# B&R Automation Studio project ACOPOStrak_DATech_Pilot (part 6)

#### Main.st
```iecst
PROGRAM _INIT
	currentProcess							:= E_PROCESS_Stage11;
	fbUserData.Axis							:= ADR(StStage[10].Shuttle);
	nextSlot 								:= ADR(StStage[11]);

	fbShuttleOutCheck.ProcessPoint			:= ADR(ptStage11);

	targetSlot ACCESS ADR(StStage[10]);
	shuttleID ACCESS ADR(interface.Trak.Data[0]);
END_PROGRAM

PROGRAM _CYCLIC
	IF gSim = TRUE THEN
		bBlockReadOnceAck := bBlockReadOnce;
		bBlockSendOnceAck := bBlockSendOnce;
		bBlockSendShuttleIDAck := bBlockSendShuttleID;

		IF interface.Trak.ShuttleArrived = TRUE THEN
			interface.Equipment.Ready 		:= FALSE;

			tmr.IN 							:= TRUE;
			tmr.PT 							:= T#1s;
		END_IF

		IF tmr.Q = TRUE THEN
			interface.Equipment.Done 		:= TRUE;
		END_IF

		IF interface.Trak.ShuttleArrived = FALSE THEN
			tmr.IN							:= FALSE;
			interface.Equipment.Ready 		:= TRUE;
			interface.Equipment.Done 		:= FALSE;
		END_IF

		tmr();
	END_IF

	IF targetSlot.Interface = E_SLOT_UNKNOWN THEN
		step 				:= 0;
	END_IF

	CASE step OF
		0:	(* Modbus Interface Initialize and Shuttle Check *)
			bBlockSendShuttleID					:= FALSE;
			bBlockSendOnce						:= FALSE;
			bBlockReadOnce						:= FALSE;

			//interface.Trak.ShuttleArrived		:= FALSE;

			IF targetSlot.Shuttle.controlif <> 0 AND bBlockSendOnceAck = FALSE AND bBlockReadOnceAck = FALSE AND bBlockSendShuttleIDAck = FALSE THEN
				step 							:= 10;
			END_IF

		10:	(* Read Shuttle Data from userData *)
			fbUserData.DataAddress 				:= ADR(userData);
			fbUserData.DataSize 				:= SIZEOF(userData);
			fbUserData.Mode						:= mcACPTRAK_USERDATA_GET;
			fbUserData.Execute 					:= TRUE;

			IF fbUserData.Done = TRUE THEN
				//End to Read Data fron user Data
				fbUserData.Execute 				:= FALSE;

				//Copy User Data to Modbus IO
				brsmemcpy(ADR(interface.Trak.Data[0]),ADR(userData.SerialNumber), 11);
				brsmemcpy(ADR(interface.Trak.Data2[0]),ADR(userData.Data[0]), SIZEOF(userData.Data));

				//Start to Write userdata to Modbus
				bBlockSendOnce					:= TRUE;
				bBlockSendShuttleID				:= TRUE;
				step 							:= 11;
			END_IF

		11: (* Check End of write to Modbus *)
			IF bBlockSendOnceAck AND bBlockSendShuttleIDAck THEN
				bBlockSendOnce					:= FALSE;
				bBlockSendShuttleID				:= FALSE;
				step							:= 20;
			END_IF

		20: (* Check Process Ready *)
			IF targetSlot.Interface = E_SLOT_PROCESS_READY THEN
				step 							:= 30;
			ELSIF targetSlot.Shuttle.controlif = 0 THEN
				step 							:= 0;
			END_IF

		30:	(* Check Assemble Status and Slot Status *)
			IF (gSts.AsmState = E_ASM_PROCESS OR gSts.AsmState = E_ASM_IDLE)
				AND targetSlot.Interface = E_SLOT_PROCESS_READY THEN
				interface.Trak.ShuttleArrived	:= TRUE;
				fbShuttleOutCheck.Enable		:= TRUE;
				step 							:= 100;
			END_IF

		100: (* Wait Proess End and Next Stage Ready *)
			IF interface.Equipment.Done = TRUE AND NextReady THEN
				//Start to Read Data from PLC
				bBlockReadOnce					:= TRUE;
				step 							:= 101;
			END_IF

		101:
			IF bBlockReadOnceAck = TRUE THEN
				// Save Current Process Status
				userData.ProcessStatus			:= currentProcess;

				// Read process data from PLC
				brsmemcpy(ADR(userData.Data[0]), ADR(interface.Equipment.Data2[0]), SIZEOF(interface.Equipment.Data2));

				// End to Read Data from PLC
				bBlockReadOnce					:= FALSE;
				step := 110;
			END_IF

		110: 	//Write User Data
			fbUserData.DataAddress 				:= ADR(userData);
			fbUserData.DataSize 				:= SIZE_OF_USERDATA;
			fbUserData.Mode						:= mcACPTRAK_USERDATA_SET;
			fbUserData.Execute 					:= TRUE;

			IF fbUserData.Done = TRUE THEN
				fbUserData.Execute 				:= FALSE;
				//	interface.Trak.ShuttleArrived 	:= FALSE;
				targetSlot.Interface 			:= E_SLOT_TAKEOUT_READY;
				targetSlot.NextStage			:= nextSlot;
				step 							:= 120;
			END_IF

		120: 	//Done Check
			IF interface.Equipment.Done = FALSE THEN
				step 						:= 0;
			END_IF
	END_CASE;

	IF fbShuttleOutCheck.EventCount > 0 THEN
		interface.Trak.ShuttleArrived	:= FALSE;
		fbShuttleOutCheck.Enable		:= FALSE;
	END_IF

	IF targetSlot.Shuttle.controlif = 0 AND shuttleID <> '' THEN
		brsmemset(ADR(interface.Trak.Data[0]),0,11);
	END_IF

	fbUserData();
	fbShuttleOutCheck();
	Timer();
	Timer2();

END_PROGRAM
```

### Program Logical/Source/Control/ifStage12 (IEC) - CCR 3

#### Main.st
```iecst
PROGRAM _INIT
	currentProcess							:= E_PROCESS_Stage12;
	fbUserData.Axis							:= ADR(StStage[11].Shuttle);
	nextSlot 								:= ADR(StStage[12]);

	fbShuttleOutCheck.ProcessPoint			:= ADR(ptStage12);

	targetSlot ACCESS ADR(StStage[11]);
	shuttleID ACCESS ADR(interface.Trak.Data[0]);
END_PROGRAM

PROGRAM _CYCLIC
	IF gSim = TRUE THEN
		bBlockReadOnceAck := bBlockReadOnce;
		bBlockSendOnceAck := bBlockSendOnce;
		bBlockSendShuttleIDAck := bBlockSendShuttleID;

		IF interface.Trak.ShuttleArrived = TRUE THEN
			interface.Equipment.Ready 		:= FALSE;

			tmr.IN 							:= TRUE;
			tmr.PT 							:= T#1s;
		END_IF

		IF tmr.Q = TRUE THEN
			interface.Equipment.Done 		:= TRUE;
		END_IF

		IF interface.Trak.ShuttleArrived = FALSE THEN
			tmr.IN							:= FALSE;
			interface.Equipment.Ready 		:= TRUE;
			interface.Equipment.Done 		:= FALSE;
		END_IF

		tmr();
	END_IF

	IF targetSlot.Interface = E_SLOT_UNKNOWN THEN
		step 				:= 0;
	END_IF

	CASE step OF
		0:	(* Modbus Interface Initialize and Shuttle Check *)
			bBlockSendShuttleID					:= FALSE;
			bBlockSendOnce						:= FALSE;
			bBlockReadOnce						:= FALSE;

			//interface.Trak.ShuttleArrived		:= FALSE;

			IF targetSlot.Shuttle.controlif <> 0 AND bBlockSendOnceAck = FALSE AND bBlockReadOnceAck = FALSE AND bBlockSendShuttleIDAck = FALSE THEN
				step 							:= 10;
			END_IF

		10:	(* Read Shuttle Data from userData *)
			fbUserData.DataAddress 				:= ADR(userData);
			fbUserData.DataSize 				:= SIZEOF(userData);
			fbUserData.Mode						:= mcACPTRAK_USERDATA_GET;
			fbUserData.Execute 					:= TRUE;

			IF fbUserData.Done = TRUE THEN
				//End to Read Data fron user Data
				fbUserData.Execute 				:= FALSE;

				//Copy User Data to Modbus IO
				brsmemcpy(ADR(interface.Trak.Data[0]),ADR(userData.SerialNumber), 11);
				brsmemcpy(ADR(interface.Trak.Data2[0]),ADR(userData.Data[0]), SIZEOF(userData.Data));

				//Start to Write userdata to Modbus
				bBlockSendOnce					:= TRUE;
				bBlockSendShuttleID				:= TRUE;
				step 							:= 11;
			END_IF

		11: (* Check End of write to Modbus *)
			IF bBlockSendOnceAck AND bBlockSendShuttleIDAck THEN
				bBlockSendOnce					:= FALSE;
				bBlockSendShuttleID				:= FALSE;
				step							:= 20;
			END_IF

		20: (* Check Process Ready *)
			IF targetSlot.Interface = E_SLOT_PROCESS_READY THEN
				step 							:= 30;
			ELSIF targetSlot.Shuttle.controlif = 0 THEN
				step 							:= 0;
			END_IF

		30:	(* Check Assemble Status and Slot Status *)
			IF (gSts.AsmState = E_ASM_PROCESS OR gSts.AsmState = E_ASM_IDLE)
				AND targetSlot.Interface = E_SLOT_PROCESS_READY THEN
				interface.Trak.ShuttleArrived	:= TRUE;
				fbShuttleOutCheck.Enable		:= TRUE;
				step 							:= 100;
			END_IF

		100: (* Wait Proess End and Next Stage Ready *)
			IF interface.Equipment.Done = TRUE AND NextReady THEN
				//Start to Read Data from PLC
				bBlockReadOnce					:= TRUE;
				step 							:= 101;
			END_IF

		101:
			IF bBlockReadOnceAck = TRUE THEN
				// Save Current Process Status
				userData.ProcessStatus			:= currentProcess;

				// Read process data from PLC
				brsmemcpy(ADR(userData.Data[0]), ADR(interface.Equipment.Data2[0]), SIZEOF(interface.Equipment.Data2));

				// End to Read Data from PLC
				bBlockReadOnce					:= FALSE;
				step := 110;
			END_IF

		110: 	//Write User Data
			fbUserData.DataAddress 				:= ADR(userData);
			fbUserData.DataSize 				:= SIZE_OF_USERDATA;
			fbUserData.Mode						:= mcACPTRAK_USERDATA_SET;
			fbUserData.Execute 					:= TRUE;

			IF fbUserData.Done = TRUE THEN
				fbUserData.Execute 				:= FALSE;
				//	interface.Trak.ShuttleArrived 	:= FALSE;
				targetSlot.Interface 			:= E_SLOT_TAKEOUT_READY;
				targetSlot.NextStage			:= nextSlot;
				step 							:= 120;
			END_IF

		120: 	//Done Check
			IF interface.Equipment.Done = FALSE THEN
				step 						:= 0;
			END_IF
	END_CASE;

	IF fbShuttleOutCheck.EventCount > 0 THEN
		interface.Trak.ShuttleArrived	:= FALSE;
		fbShuttleOutCheck.Enable		:= FALSE;
	END_IF

	IF targetSlot.Shuttle.controlif = 0 AND shuttleID <> '' THEN
		brsmemset(ADR(interface.Trak.Data[0]),0,11);
	END_IF

	fbUserData();
	fbShuttleOutCheck();
	Timer();
	Timer2();

END_PROGRAM
```

### Program Logical/Source/Control/if3D (IEC) - 3D scanner flying 

#### Main.st - Init, cyclic, exit code
```iecst
PROGRAM _INIT

	fbFlyStage.InPoint				:= ADR(pt3DIn);
	fbFlyStage.OutPoint				:= ADR(pt3DOut);
	fbFlyStage.MaximumShuttleCount	:= 1;
	fbFlyStage.InitShuttleCount		:= 1;

	fbTrig.ProcessPoint				:= ADR(pt3D);
	fbTrigInfo.ProcessPoint			:= ADR(pt3D);

	ShReadInfo.Axis	:= ADR(Axis);

	ShReadSectorPosInfo.Sector		:= ADR(SectorTrackAll);
	ShReadSectorPosInfo.Axis		:= ADR(Axis);

	fbUserData.Axis	:= ADR(fbTrigInfo.TrgPointInfo);

	shuttleID ACCESS ADR(interface.Trak.Data[0]);

	g3DStartPos	:= 10.52;
	g3DEndPos	:= 10.588;
	AddedTime	:= 14000; //140000

END_PROGRAM

PROGRAM _CYCLIC

	bModuleOK;
	bMovQuitFifoEmpty;
	bMovQuitFifoFull;
	bMovQuitTargetTimeVioloation;
	bMovQuitMaxFrequencyViolation;

	//////////////////////////////////////////////////////////////////////////////////
	// 3D scanner with DS1119 module
	//////////////////////////////////////////////////////////////////////////////////
//	MovTargetTime	:= MovTimeValid + AddedTime;

	IF gSts.AsmState = E_ASM_EMS OR gSts.AsmState = E_ASM_IDLE OR gSts.AsmState = E_ASM_INITIALIZATION THEN
		//	fbFlyStage.Enable	:= FALSE;
		Step				:= STEP_WAIT;
	ELSIF gSts.AsmState = E_ASM_PROCESS OR gSts.AsmState = E_ASM_MANUAL OR gSts.AsmState = E_ASM_ON THEN
		//	fbFlyStage.Enable	:= TRUE;
	END_IF

	CASE Step OF

		STEP_WAIT:
			IF fbTrigInfo.TrgPointInfo.Axis.controlif = 0 AND shuttleID <> '' THEN
				brsmemset(ADR(interface.Trak.Data[0]), 0, 11);
				userData.SerialNumber	:= '';
			END_IF

			interface.Trak.ShuttleArrived	:= FALSE;
			doTrigger						:= FALSE;
//			EncCnt							:= 0;
			IF gSts.AsmState = E_ASM_PROCESS OR gSts.AsmState = E_ASM_MANUAL OR gSts.AsmState = E_ASM_ON THEN
				fbTrig.Enable	:= TRUE;

				IF fbTrig.Valid THEN
					MovTargetPosition	:= LREAL_TO_DINT((g3DStartPos - 0.005) * 1000000);
					Step				:= STEP_IDLE;
				END_IF
			ELSE
				fbTrig.Enable	:= FALSE;
			END_IF

		STEP_IDLE:

			IF fbTrig.EventCount > 0 THEN
				fbTrigInfo.Execute	:= TRUE;

				fbUserData.DataAddress	:= ADR(userData);
				fbUserData.DataSize		:= SIZE_OF_USERDATA;
				fbUserData.Mode			:= mcACPTRAK_USERDATA_GET;
				fbUserData.Execute		:= TRUE;

				Step					:= STEP_GETSH;
			END_IF

		STEP_GETSH:
			IF fbTrigInfo.Done AND fbUserData.Done THEN
				interface.Trak.ShuttleArrived	:= TRUE;
				Axis							:= fbTrigInfo.TrgPointInfo.Axis;

				brsmemcpy(ADR(interface.Trak.Data[0]), ADR(userData.SerialNumber), 11);

				ShReadSectorPosInfo.Enable		:= TRUE;

				IF ShReadSectorPosInfo.Valid THEN
					Step			:= STEP_PRERUN;
					MovTargetTime	:= MovTimeValid + AddedTime;
				END_IF
			END_IF

		STEP_PRERUN:
			MovEnable			:= TRUE;
			MovTargetPosition	:= LREAL_TO_DINT((g3DStartPos - 0.005) * 1000000);
			MovTargetTime 		:= MovTargetTime + 2000;

			IF ShReadSectorPosInfo.Info.Position >= g3DStartPos - 0.005 THEN
				doTrigger	:= TRUE;
				Step		:= STEP_END;
			END_IF

//			IF EncCnt >= 1 THEN
//				IF ShReadSectorPosInfo.Info.Position < g3DStartPos - 0.005 THEN
//					MovTargetPosition	:= LREAL_TO_DINT((g3DStartPos - 0.005) * 1000000);
//				ELSE
//					MovTargetPosition	:= LREAL_TO_DINT((g3DStartPos - 0.005) * 1000000);
//				END_IF
//			END_IF
			//			EncCnt	:= EncCnt + 1;
//			MovEnable			:= TRUE;
//			MovTargetPosition	:= LREAL_TO_DINT(ShReadSectorPosInfo.Info.Position * 1000000);
			//			IF ShReadSectorPosInfo.Info.Position >= g3DStartPos THEN
//				doTrigger	:= TRUE;
//				Step		:= STEP_END;
//			END_IF

		STEP_END:
			MovTargetPosition	:= LREAL_TO_DINT(ShReadSectorPosInfo.Info.Position * 1000000);
			MovTargetTime 		:= MovTargetTime + 2000;

			IF ShReadSectorPosInfo.Info.Position >= g3DEndPos THEN
				ShReadSectorPosInfo.Enable		:= FALSE;
				interface.Trak.ShuttleArrived	:= FALSE;
				MovEnable						:= FALSE;
				doTrigger						:= FALSE;
				fbTrigInfo.Execute				:= FALSE;
				fbUserData.Execute				:= FALSE;
				Step							:= STEP_WAIT;
			END_IF

	END_CASE;

	// FB calls
	fbFlyStage();
	fbTrig();
	fbTrigInfo();
	fbUserData();
	ShReadSectorPosInfo();

END_PROGRAM
```

#### Variables.var - Local variables
```iecst
(**)
VAR
	MovEnable : BOOL;
	MovReset : BOOL;
	MovTargetPosition : DINT;
	MovTargetTime : DINT;
	MovPosition : DINT;
	MovTimeValid : DINT;
	AddedTime : DINT;
END_VAR
(**)
VAR
	nextReady : BOOL;
	shuttleID : REFERENCE TO STRING[19];
	userData : ShuttleUserData_typ;
	fbUserData : MC_BR_ShCopyUserData_AcpTrak;
END_VAR
(**)
VAR
	interface : Interface_Process_1Sh;
	fbFlyStage : MyTrak_TicketArea;
END_VAR
(**)
VAR
	fbTrigInfo : MC_BR_TrgPointGetInfo_AcpTrak;
	fbTrig : MC_BR_TrgPointEnable_AcpTrak;
	Axis : McAxisType;
	ShReadInfo : MC_BR_ShReadInfo_AcpTrak;
	ShReadSectorPosInfo : MC_BR_ShReadSectorPos_AcpTrak;
	Step : STEP_3DSensor;
	doTrigger : BOOL;
END_VAR
(**)
VAR
	timeMeasurement : TimingMeasurement_type;
END_VAR
(**)
VAR
	MoveTime : REAL;
	EncCnt : UINT;
END_VAR
(*Monitoring*)
VAR
	bModuleOK : BOOL;
	bMovQuitFifoEmpty : BOOL;
	bMovQuitFifoFull : BOOL;
	bMovQuitTargetTimeVioloation : BOOL;
	bMovQuitMaxFrequencyViolation : BOOL;
END_VAR
```

#### Types.typ
```iecst
TYPE
	STEP_3DSensor :
		(
		STEP_WAIT := 0,
		STEP_IDLE := 1,
		STEP_GETSH := 2,
		STEP_PRERUN := 3,
		STEP_END := 4
		);
	TimingMeasurement_type : 	STRUCT
		NextShuttle : MyTime_TimeCheck;
		ProcessingTime : MyTime_TimeCheck;
		MovementTime : MyTime_TimeCheck;
	END_STRUCT;
END_TYPE
```

### Program Logical/Source/Control/ifStage13 (IEC) - CCR 3

#### Main.st
```iecst
PROGRAM _INIT
	currentProcess							:= E_PROCESS_Stage13;
	fbUserData.Axis							:= ADR(StStage[12].Shuttle);
	nextSlot 								:= ADR(StStage[13]);

	fbShuttleOutCheck.ProcessPoint			:= ADR(ptStage13);

	targetSlot ACCESS ADR(StStage[12]);
	shuttleID ACCESS ADR(interface.Trak.Data[0]);

	NextReady 								:= TRUE;
END_PROGRAM

PROGRAM _CYCLIC
	IF gSim = TRUE THEN
		bBlockReadOnceAck := bBlockReadOnce;
		bBlockSendOnceAck := bBlockSendOnce;
		bBlockSendShuttleIDAck := bBlockSendShuttleID;

		IF interface.Trak.ShuttleArrived = TRUE THEN
			interface.Equipment.Ready 		:= FALSE;

			tmr.IN 							:= TRUE;
			tmr.PT 							:= T#1s;
		END_IF

		IF tmr.Q = TRUE THEN
			interface.Equipment.Done 		:= TRUE;
		END_IF

		IF interface.Trak.ShuttleArrived = FALSE THEN
			tmr.IN							:= FALSE;
			interface.Equipment.Ready 		:= TRUE;
			interface.Equipment.Done 		:= FALSE;
		END_IF

		tmr();
	END_IF

	IF targetSlot.Interface = E_SLOT_UNKNOWN THEN
		step 				:= 0;
	END_IF

	CASE step OF
		0:	(* Modbus Interface Initialize and Shuttle Check *)
			bBlockSendShuttleID					:= FALSE;
			bBlockSendOnce						:= FALSE;
			bBlockReadOnce						:= FALSE;

			//interface.Trak.ShuttleArrived		:= FALSE;

			IF targetSlot.Shuttle.controlif <> 0 AND bBlockSendOnceAck = FALSE AND bBlockReadOnceAck = FALSE AND bBlockSendShuttleIDAck = FALSE THEN
				step 							:= 10;
			END_IF

		10:	(* Read Shuttle Data from userData *)
			fbUserData.DataAddress 				:= ADR(userData);
			fbUserData.DataSize 				:= SIZEOF(userData);
			fbUserData.Mode						:= mcACPTRAK_USERDATA_GET;
			fbUserData.Execute 					:= TRUE;

			IF fbUserData.Done = TRUE THEN
				//End to Read Data fron user Data
				fbUserData.Execute 				:= FALSE;

				//Copy User Data to Modbus IO
				brsmemcpy(ADR(interface.Trak.Data[0]),ADR(userData.SerialNumber), 11);
				brsmemcpy(ADR(interface.Trak.Data2[0]),ADR(userData.Data[0]), SIZEOF(userData.Data));

				//Start to Write userdata to Modbus
				bBlockSendOnce					:= TRUE;
				bBlockSendShuttleID				:= TRUE;
				step 							:= 11;
			END_IF

		11: (* Check End of write to Modbus *)
			IF bBlockSendOnceAck AND bBlockSendShuttleIDAck THEN
				bBlockSendOnce					:= FALSE;
				bBlockSendShuttleID				:= FALSE;
				step							:= 20;
			END_IF

		20: (* Check Process Ready *)
			IF targetSlot.Interface = E_SLOT_PROCESS_READY THEN
				step 							:= 30;
			ELSIF targetSlot.Shuttle.controlif = 0 THEN
				step 							:= 0;
			END_IF

		30:	(* Check Assemble Status and Slot Status *)
			IF (gSts.AsmState = E_ASM_PROCESS OR gSts.AsmState = E_ASM_IDLE)
				AND targetSlot.Interface = E_SLOT_PROCESS_READY THEN
				interface.Trak.ShuttleArrived	:= TRUE;
				fbShuttleOutCheck.Enable		:= TRUE;
				step 							:= 100;
			END_IF

		100: (* Wait Proess End and Next Stage Ready *)
			IF interface.Equipment.Done = TRUE AND NextReady THEN
				//Start to Read Data from PLC
				bBlockReadOnce					:= TRUE;
				step 							:= 101;
			END_IF

		101:
			IF bBlockReadOnceAck = TRUE THEN
				// Save Current Process Status
				userData.ProcessStatus			:= currentProcess;

				// Read process data from PLC
				brsmemcpy(ADR(userData.Data[0]), ADR(interface.Equipment.Data2[0]), SIZEOF(interface.Equipment.Data2));

				// End to Read Data from PLC
				bBlockReadOnce					:= FALSE;
				step := 110;
			END_IF

		110: 	//Write User Data
			fbUserData.DataAddress 				:= ADR(userData);
			fbUserData.DataSize 				:= SIZE_OF_USERDATA;
			fbUserData.Mode						:= mcACPTRAK_USERDATA_SET;
			fbUserData.Execute 					:= TRUE;

			IF fbUserData.Done = TRUE THEN
				fbUserData.Execute 				:= FALSE;
				//	interface.Trak.ShuttleArrived 	:= FALSE;
				targetSlot.Interface 			:= E_SLOT_TAKEOUT_READY;
				targetSlot.NextStage			:= nextSlot;
				step 							:= 120;
			END_IF

		120: 	//Done Check
			IF interface.Equipment.Done = FALSE THEN
				step 						:= 0;
			END_IF
	END_CASE;

	IF fbShuttleOutCheck.EventCount > 0 THEN
		interface.Trak.ShuttleArrived	:= FALSE;
		fbShuttleOutCheck.Enable		:= FALSE;
	END_IF

	IF targetSlot.Shuttle.controlif = 0 AND shuttleID <> '' THEN
		brsmemset(ADR(interface.Trak.Data[0]),0,11);
	END_IF

	fbUserData();
	fbShuttleOutCheck();
	Timer();
	Timer2();

END_PROGRAM
```

### Program Logical/Source/Control/ifStage14 (IEC) - CSZ

#### Variables.var
```iecst
(**)
VAR
	currentProcess : E_PROCESS_STATUS;
	targetSlot : REFERENCE TO MyTrakSlotType;
	nextSlot : {REDUND_UNREPLICABLE} UDINT;
	shuttleID : REFERENCE TO STRING[19];
END_VAR
(**)
VAR
	step : DINT;
END_VAR
(**)
VAR
	interface : Interface_Process;
	userData : ShuttleUserData_typ;
END_VAR
(**)
VAR
	fbUserData : MC_BR_ShCopyUserData_AcpTrak;
END_VAR
(**)
VAR
	tmr : TON;
	fbShuttleOutCheck : MC_BR_TrgPointEnable_AcpTrak;
END_VAR
(**)
VAR
	NextReady : BOOL;
	Timer : TON;
	Timer2 : TON;
END_VAR
(**)
VAR
	bBlockSendOnce : BOOL;
	bBlockSendOnceAck : BOOL;
	bBlockReadOnce : BOOL;
	bBlockReadOnceAck : BOOL;
	bBlockSendShuttleID : BOOL;
	bBlockSendShuttleIDAck : BOOL;
END_VAR
(**)
VAR
	fbInterLock : MC_BR_BarrierCommand_AcpTrak;
	fbBarReadInfo : MC_BR_BarrierReadInfo_AcpTrak;
	ptInterlock : UDINT;
END_VAR
```

#### Main.st
```iecst
PROGRAM _INIT
	currentProcess							:= E_PROCESS_Stage14;
	fbUserData.Axis							:= ADR(StStage[13].Shuttle);
	nextSlot 								:= ADR(StStage[14]);

	fbShuttleOutCheck.ProcessPoint			:= ADR(ptStage14);

	ptInterlock								:= ADR(ptCSZInt);

	targetSlot ACCESS ADR(StStage[13]);
	shuttleID ACCESS ADR(interface.Trak.Data[0]);
END_PROGRAM

PROGRAM _CYCLIC
	IF gSim = TRUE THEN
		bBlockReadOnceAck := bBlockReadOnce;
		bBlockSendOnceAck := bBlockSendOnce;
		bBlockSendShuttleIDAck := bBlockSendShuttleID;

		IF interface.Trak.ShuttleArrived = TRUE THEN
			interface.Equipment.Ready 		:= FALSE;

			tmr.IN 							:= TRUE;
			tmr.PT 							:= T#1s;
		END_IF

		IF tmr.Q = TRUE THEN
			interface.Equipment.Done 		:= TRUE;
		END_IF

		IF interface.Trak.ShuttleArrived = FALSE THEN
			tmr.IN							:= FALSE;
			interface.Equipment.Ready 		:= TRUE;
			interface.Equipment.Done 		:= FALSE;
		END_IF

		tmr();
	END_IF

	//-----------------INTERLOCK--------------------
//	IF fbInterLock.Done = TRUE OR fbInterLock.Busy = TRUE OR fbInterLock.Error = TRUE THEN
//		fbInterLock.Execute 	:= FALSE;
//	ELSIF interface.Equipment.Ready = FALSE AND fbBarReadInfo.BarrierInfo.Status <> mcACPTRAK_BARRIER_CLOSED THEN
//		fbInterLock.Command 	:= mcACPTRAK_BARRIER_CLOSE;
//		fbInterLock.Execute 	:= TRUE;
//	ELSIF  interface.Equipment.Ready = TRUE AND fbBarReadInfo.BarrierInfo.Status <> mcACPTRAK_BARRIER_OPENED THEN
//		fbInterLock.Command 	:= mcACPTRAK_BARRIER_OPEN;
//		fbInterLock.Execute 	:= TRUE;
//	END_IF
//
//	fbBarReadInfo.Enable := TRUE;
//	fbBarReadInfo(ProcessPoint := ptInterlock);
//	fbInterLock(ProcessPoint := ptInterlock);
	//-----------------INTERLOCK--------------------

	IF targetSlot.Interface = E_SLOT_UNKNOWN THEN
		step 				:= 0;
	END_IF

	CASE step OF
		0:	(* Modbus Interface Initialize and Shuttle Check *)
			bBlockSendShuttleID					:= FALSE;
			bBlockSendOnce						:= FALSE;
			bBlockReadOnce						:= FALSE;

			//interface.Trak.ShuttleArrived		:= FALSE;

			IF targetSlot.Shuttle.controlif <> 0 AND bBlockSendOnceAck = FALSE AND bBlockReadOnceAck = FALSE AND bBlockSendShuttleIDAck = FALSE THEN
				step 							:= 10;
			END_IF

		10:	(* Read Shuttle Data from userData *)
			fbUserData.DataAddress 				:= ADR(userData);
			fbUserData.DataSize 				:= SIZEOF(userData);
			fbUserData.Mode						:= mcACPTRAK_USERDATA_GET;
			fbUserData.Execute 					:= TRUE;

			IF fbUserData.Done = TRUE THEN
				//End to Read Data fron user Data
				fbUserData.Execute 				:= FALSE;

				//Copy User Data to Modbus IO
				brsmemcpy(ADR(interface.Trak.Data[0]),ADR(userData.SerialNumber), 11);
				brsmemcpy(ADR(interface.Trak.Data2[0]),ADR(userData.Data[0]), SIZEOF(userData.Data));

				//Start to Write userdata to Modbus
				bBlockSendOnce					:= TRUE;
				bBlockSendShuttleID				:= TRUE;
				step 							:= 11;
			END_IF

		11: (* Check End of write to Modbus *)
			IF bBlockSendOnceAck AND bBlockSendShuttleIDAck THEN
				bBlockSendOnce					:= FALSE;
				bBlockSendShuttleID				:= FALSE;
				step							:= 20;
			END_IF

		20: (* Check Process Ready *)
			IF targetSlot.Interface = E_SLOT_PROCESS_READY THEN
				step 							:= 30;
			ELSIF targetSlot.Shuttle.controlif = 0 THEN
				step 							:= 0;
			END_IF

		30:	(* Check Assemble Status and Slot Status *)
			IF (gSts.AsmState = E_ASM_PROCESS OR gSts.AsmState = E_ASM_IDLE)
				AND targetSlot.Interface = E_SLOT_PROCESS_READY THEN
				interface.Trak.ShuttleArrived	:= TRUE;
				fbShuttleOutCheck.Enable		:= TRUE;
				step 							:= 100;
			END_IF

		100: (* Wait Proess End and Next Stage Ready *)
			IF interface.Equipment.Done = TRUE AND NextReady THEN
				//Start to Read Data from PLC
				bBlockReadOnce					:= TRUE;
				step 							:= 101;
			END_IF

		101:
			IF bBlockReadOnceAck = TRUE THEN
				// Save Current Process Status
				userData.ProcessStatus			:= currentProcess;

				// Read process data from PLC
				brsmemcpy(ADR(userData.Data[0]), ADR(interface.Equipment.Data2[0]), SIZEOF(interface.Equipment.Data2));

				// End to Read Data from PLC
				bBlockReadOnce					:= FALSE;
				step := 110;
			END_IF

		110: 	//Write User Data
			fbUserData.DataAddress 				:= ADR(userData);
			fbUserData.DataSize 				:= SIZE_OF_USERDATA;
			fbUserData.Mode						:= mcACPTRAK_USERDATA_SET;
			fbUserData.Execute 					:= TRUE;

			IF fbUserData.Done = TRUE THEN
				fbUserData.Execute 				:= FALSE;
				//	interface.Trak.ShuttleArrived 	:= FALSE;
				targetSlot.Interface 			:= E_SLOT_TAKEOUT_READY;
				targetSlot.NextStage			:= nextSlot;
				step 							:= 120;
			END_IF

		120: 	//Done Check
			IF interface.Equipment.Done = FALSE THEN
				step 						:= 0;
			END_IF
	END_CASE;

	IF fbShuttleOutCheck.EventCount > 0 THEN
		interface.Trak.ShuttleArrived	:= FALSE;
		fbShuttleOutCheck.Enable		:= FALSE;
	END_IF

	IF targetSlot.Shuttle.controlif = 0 AND shuttleID <> '' THEN
		brsmemset(ADR(interface.Trak.Data[0]),0,11);
	END_IF

	fbUserData();
	fbShuttleOutCheck();
	Timer();
	Timer2();

END_PROGRAM
```

### Program Logical/Source/Control/ifStage15 (IEC) - 3D arrive position

#### Main.st
```iecst
PROGRAM _INIT
	currentProcess							:= E_PROCESS_Stage15;
	fbUserData.Axis							:= ADR(StStage[14].Shuttle);
	nextSlot 								:= ADR(StStage[15]);

	fbShuttleOutCheck.ProcessPoint			:= ADR(ptStage15);

	targetSlot ACCESS ADR(StStage[14]);
	shuttleID ACCESS ADR(interface.Trak.Data[0]);
END_PROGRAM

PROGRAM _CYCLIC
	IF gSim = TRUE THEN
		bBlockReadOnceAck := bBlockReadOnce;
		bBlockSendOnceAck := bBlockSendOnce;
		bBlockSendShuttleIDAck := bBlockSendShuttleID;

		IF interface.Trak.ShuttleArrived = TRUE THEN
			interface.Equipment.Ready 		:= FALSE;

			tmr.IN 							:= TRUE;
			tmr.PT 							:= T#1s;
		END_IF

		IF tmr.Q = TRUE THEN
			interface.Equipment.Done 		:= TRUE;
		END_IF

		IF interface.Trak.ShuttleArrived = FALSE THEN
			tmr.IN							:= FALSE;
			interface.Equipment.Ready 		:= TRUE;
			interface.Equipment.Done 		:= FALSE;
		END_IF

		tmr();
	END_IF

	IF targetSlot.Interface = E_SLOT_UNKNOWN THEN
		step 				:= 0;
	END_IF

	CASE step OF
		0:	(* Modbus Interface Initialize and Shuttle Check *)
			bBlockSendShuttleID					:= FALSE;
			bBlockSendOnce						:= FALSE;
			bBlockReadOnce						:= FALSE;

			//interface.Trak.ShuttleArrived		:= FALSE;

			IF targetSlot.Shuttle.controlif <> 0 AND bBlockSendOnceAck = FALSE AND bBlockReadOnceAck = FALSE AND bBlockSendShuttleIDAck = FALSE THEN
				step 							:= 10;
			END_IF

		10:	(* Read Shuttle Data from userData *)
			fbUserData.DataAddress 				:= ADR(userData);
			fbUserData.DataSize 				:= SIZEOF(userData);
			fbUserData.Mode						:= mcACPTRAK_USERDATA_GET;
			fbUserData.Execute 					:= TRUE;

			IF fbUserData.Done = TRUE THEN
				//End to Read Data fron user Data
				fbUserData.Execute 				:= FALSE;

				//Copy User Data to Modbus IO
				brsmemcpy(ADR(interface.Trak.Data[0]),ADR(userData.SerialNumber), 11);
				brsmemcpy(ADR(interface.Trak.Data2[0]),ADR(userData.Data[0]), SIZEOF(userData.Data));

				//Start to Write userdata to Modbus
				bBlockSendOnce					:= TRUE;
				bBlockSendShuttleID				:= TRUE;
				step 							:= 11;
			END_IF

		11: (* Check End of write to Modbus *)
			IF bBlockSendOnceAck AND bBlockSendShuttleIDAck THEN
				bBlockSendOnce					:= FALSE;
				bBlockSendShuttleID				:= FALSE;
				step							:= 20;
			END_IF

		20: (* Check Process Ready *)
			IF targetSlot.Interface = E_SLOT_PROCESS_READY THEN
				step 							:= 30;
			ELSIF targetSlot.Shuttle.controlif = 0 THEN
				step 							:= 0;
			END_IF

		30:	(* Check Assemble Status and Slot Status *)
			IF (gSts.AsmState = E_ASM_PROCESS OR gSts.AsmState = E_ASM_IDLE)
				AND targetSlot.Interface = E_SLOT_PROCESS_READY THEN
				interface.Trak.ShuttleArrived	:= TRUE;
				fbShuttleOutCheck.Enable		:= TRUE;
				step 							:= 100;
			END_IF

		100: (* Wait Proess End and Next Stage Ready *)
			IF interface.Equipment.Done = TRUE AND NextReady THEN
				//Start to Read Data from PLC
				bBlockReadOnce					:= TRUE;
				step 							:= 101;
			END_IF

		101:
			IF bBlockReadOnceAck = TRUE THEN
				// Save Current Process Status
				userData.ProcessStatus			:= currentProcess;

				// Read process data from PLC
				brsmemcpy(ADR(userData.Data[0]), ADR(interface.Equipment.Data2[0]), SIZEOF(interface.Equipment.Data2));

				// End to Read Data from PLC
				bBlockReadOnce					:= FALSE;
				step := 110;
			END_IF

		110: 	//Write User Data
			fbUserData.DataAddress 				:= ADR(userData);
			fbUserData.DataSize 				:= SIZE_OF_USERDATA;
			fbUserData.Mode						:= mcACPTRAK_USERDATA_SET;
			fbUserData.Execute 					:= TRUE;

			IF fbUserData.Done = TRUE THEN
				fbUserData.Execute 				:= FALSE;
				//	interface.Trak.ShuttleArrived 	:= FALSE;
				targetSlot.Interface 			:= E_SLOT_TAKEOUT_READY;
				targetSlot.NextStage			:= nextSlot;
				step 							:= 120;
			END_IF

		120: 	//Done Check
			IF interface.Equipment.Done = FALSE THEN
				step 						:= 0;
			END_IF
	END_CASE;

	IF fbShuttleOutCheck.EventCount > 0 THEN
		interface.Trak.ShuttleArrived	:= FALSE;
		fbShuttleOutCheck.Enable		:= FALSE;
	END_IF

	IF targetSlot.Shuttle.controlif = 0 AND shuttleID <> '' THEN
		brsmemset(ADR(interface.Trak.Data[0]),0,11);
	END_IF

	fbUserData();
	fbShuttleOutCheck();
	Timer();
	Timer2();

END_PROGRAM
```

### Program Logical/Source/Control/ifStage16 (IEC) - Diameter inspection

#### Variables.var
```iecst
(**)
VAR
	currentProcess : E_PROCESS_STATUS;
	targetSlot : REFERENCE TO MyTrakSlotType;
	nextSlot : {REDUND_UNREPLICABLE} UDINT;
	shuttleID : REFERENCE TO STRING[19];
END_VAR
(**)
VAR
	step : DINT;
END_VAR
(**)
VAR
	interface : Interface_Process;
	userData : ShuttleUserData_typ;
END_VAR
(**)
VAR
	fbUserData : MC_BR_ShCopyUserData_AcpTrak;
END_VAR
(**)
VAR
	tmr : TON;
	fbShuttleOutCheck : MC_BR_TrgPointEnable_AcpTrak;
END_VAR
(**)
VAR
	NextReady : BOOL;
	Timer : TON;
	Timer2 : TON;
END_VAR
(**)
VAR
	bBlockSendOnce : BOOL;
	bBlockSendOnceAck : BOOL;
	bBlockReadOnce : BOOL;
	bBlockReadOnceAck : BOOL;
	bBlockSendShuttleID : BOOL;
	bBlockSendShuttleIDAck : BOOL;
END_VAR
```

#### Main.st
```iecst
PROGRAM _INIT
	currentProcess							:= E_PROCESS_Stage16;
	fbUserData.Axis							:= ADR(StStage[15].Shuttle);
	nextSlot 								:= ADR(StStage[16]);

	fbShuttleOutCheck.ProcessPoint			:= ADR(ptStage16);

	targetSlot ACCESS ADR(StStage[15]);
	shuttleID ACCESS ADR(interface.Trak.Data[0]);
END_PROGRAM

PROGRAM _CYCLIC
	IF gSim = TRUE THEN
		bBlockReadOnceAck := bBlockReadOnce;
		bBlockSendOnceAck := bBlockSendOnce;
		bBlockSendShuttleIDAck := bBlockSendShuttleID;

		IF interface.Trak.ShuttleArrived = TRUE THEN
			interface.Equipment.Ready 		:= FALSE;

			tmr.IN 							:= TRUE;
			tmr.PT 							:= T#1s;
		END_IF

		IF tmr.Q = TRUE THEN
			interface.Equipment.Done 		:= TRUE;
		END_IF

		IF interface.Trak.ShuttleArrived = FALSE THEN
			tmr.IN							:= FALSE;
			interface.Equipment.Ready 		:= TRUE;
			interface.Equipment.Done 		:= FALSE;
		END_IF

		tmr();
	END_IF

	IF targetSlot.Interface = E_SLOT_UNKNOWN THEN
		step 				:= 0;
	END_IF

	CASE step OF
		0:	(* Modbus Interface Initialize and Shuttle Check *)
			bBlockSendShuttleID					:= FALSE;
			bBlockSendOnce						:= FALSE;
			bBlockReadOnce						:= FALSE;

			//interface.Trak.ShuttleArrived		:= FALSE;

			IF targetSlot.Shuttle.controlif <> 0 AND bBlockSendOnceAck = FALSE AND bBlockReadOnceAck = FALSE AND bBlockSendShuttleIDAck = FALSE THEN
				step 							:= 10;
			END_IF

		10:	(* Read Shuttle Data from userData *)
			fbUserData.DataAddress 				:= ADR(userData);
			fbUserData.DataSize 				:= SIZEOF(userData);
			fbUserData.Mode						:= mcACPTRAK_USERDATA_GET;
			fbUserData.Execute 					:= TRUE;

			IF fbUserData.Done = TRUE THEN
				//End to Read Data fron user Data
				fbUserData.Execute 				:= FALSE;

				//Copy User Data to Modbus IO
				brsmemcpy(ADR(interface.Trak.Data[0]),ADR(userData.SerialNumber), 11);
				brsmemcpy(ADR(interface.Trak.Data2[0]),ADR(userData.Data[0]), SIZEOF(userData.Data));

				//Start to Write userdata to Modbus
				bBlockSendOnce					:= TRUE;
				bBlockSendShuttleID				:= TRUE;
				step 							:= 11;
			END_IF

		11: (* Check End of write to Modbus *)
			IF bBlockSendOnceAck AND bBlockSendShuttleIDAck THEN
				bBlockSendOnce					:= FALSE;
				bBlockSendShuttleID				:= FALSE;
				step							:= 20;
			END_IF

		20: (* Check Process Ready *)
			IF targetSlot.Interface = E_SLOT_PROCESS_READY THEN
				step 							:= 30;
			ELSIF targetSlot.Shuttle.controlif = 0 THEN
				step 							:= 0;
			END_IF

		30:	(* Check Assemble Status and Slot Status *)
			IF (gSts.AsmState = E_ASM_PROCESS OR gSts.AsmState = E_ASM_IDLE)
				AND targetSlot.Interface = E_SLOT_PROCESS_READY THEN
				interface.Trak.ShuttleArrived	:= TRUE;
				fbShuttleOutCheck.Enable		:= TRUE;
				step 							:= 100;
			END_IF

		100: (* Wait Proess End and Next Stage Ready *)
			IF interface.Equipment.Done = TRUE AND NextReady THEN
				//Start to Read Data from PLC
				bBlockReadOnce					:= TRUE;
				step 							:= 101;
			END_IF

		101:
			IF bBlockReadOnceAck = TRUE THEN
				// Save Current Process Status
				userData.ProcessStatus			:= currentProcess;

				// Read process data from PLC
				brsmemcpy(ADR(userData.Data[0]), ADR(interface.Equipment.Data2[0]), SIZEOF(interface.Equipment.Data2));

				// End to Read Data from PLC
				bBlockReadOnce					:= FALSE;
				step := 110;
			END_IF

		110: 	//Write User Data
			fbUserData.DataAddress 				:= ADR(userData);
			fbUserData.DataSize 				:= SIZE_OF_USERDATA;
			fbUserData.Mode						:= mcACPTRAK_USERDATA_SET;
			fbUserData.Execute 					:= TRUE;

			IF fbUserData.Done = TRUE THEN
				fbUserData.Execute 				:= FALSE;
				//	interface.Trak.ShuttleArrived 	:= FALSE;
				targetSlot.Interface 			:= E_SLOT_TAKEOUT_READY;
				targetSlot.NextStage			:= nextSlot;
				step 							:= 120;
			END_IF

		120: 	//Done Check
			IF interface.Equipment.Done = FALSE THEN
				step 						:= 0;
			END_IF
	END_CASE;

	IF fbShuttleOutCheck.EventCount > 0 THEN
		interface.Trak.ShuttleArrived	:= FALSE;
		fbShuttleOutCheck.Enable		:= FALSE;
	END_IF

	IF targetSlot.Shuttle.controlif = 0 AND shuttleID <> '' THEN
		brsmemset(ADR(interface.Trak.Data[0]),0,11);
	END_IF

	fbUserData();
	fbShuttleOutCheck();
	Timer();
	Timer2();

END_PROGRAM
```

### Program Logical/Source/Control/ifStage17 (IEC) - NG out

#### Main.st
```iecst
PROGRAM _INIT
	currentProcess							:= E_PROCESS_Stage17;
	fbUserData.Axis							:= ADR(StStage[16].Shuttle);
	nextSlot 								:= ADR(StStage[17]);

	fbShuttleOutCheck.ProcessPoint			:= ADR(ptStage17);

	targetSlot ACCESS ADR(StStage[16]);
	shuttleID ACCESS ADR(interface.Trak.Data[0]);
END_PROGRAM

PROGRAM _CYCLIC
	IF gSim = TRUE THEN
		bBlockReadOnceAck := bBlockReadOnce;
		bBlockSendOnceAck := bBlockSendOnce;
		bBlockSendShuttleIDAck := bBlockSendShuttleID;

		IF interface.Trak.ShuttleArrived = TRUE THEN
			interface.Equipment.Ready 		:= FALSE;

			tmr.IN 							:= TRUE;
			tmr.PT 							:= T#1s;
		END_IF

		IF tmr.Q = TRUE THEN
			interface.Equipment.Done 		:= TRUE;
		END_IF

		IF interface.Trak.ShuttleArrived = FALSE THEN
			tmr.IN							:= FALSE;
			interface.Equipment.Ready 		:= TRUE;
			interface.Equipment.Done 		:= FALSE;
		END_IF

		tmr();
	END_IF

	IF targetSlot.Interface = E_SLOT_UNKNOWN THEN
		step 				:= 0;
	END_IF

	CASE step OF
		0:	(* Modbus Interface Initialize and Shuttle Check *)
			bBlockSendShuttleID					:= FALSE;
			bBlockSendOnce						:= FALSE;
			bBlockReadOnce						:= FALSE;

			//interface.Trak.ShuttleArrived		:= FALSE;

			IF targetSlot.Shuttle.controlif <> 0 AND bBlockSendOnceAck = FALSE AND bBlockReadOnceAck = FALSE AND bBlockSendShuttleIDAck = FALSE THEN
				step 							:= 10;
			END_IF

		10:	(* Read Shuttle Data from userData *)
			fbUserData.DataAddress 				:= ADR(userData);
			fbUserData.DataSize 				:= SIZEOF(userData);
			fbUserData.Mode						:= mcACPTRAK_USERDATA_GET;
			fbUserData.Execute 					:= TRUE;

			IF fbUserData.Done = TRUE THEN
				//End to Read Data fron user Data
				fbUserData.Execute 				:= FALSE;

				//Copy User Data to Modbus IO
				brsmemcpy(ADR(interface.Trak.Data[0]),ADR(userData.SerialNumber), 11);
				brsmemcpy(ADR(interface.Trak.Data2[0]),ADR(userData.Data[0]), SIZEOF(userData.Data));

				//Start to Write userdata to Modbus
				bBlockSendOnce					:= TRUE;
				bBlockSendShuttleID				:= TRUE;
				step 							:= 11;
			END_IF

		11: (* Check End of write to Modbus *)
			IF bBlockSendOnceAck AND bBlockSendShuttleIDAck THEN
				bBlockSendOnce					:= FALSE;
				bBlockSendShuttleID				:= FALSE;
				step							:= 20;
			END_IF

		20: (* Check Process Ready *)
			IF targetSlot.Interface = E_SLOT_PROCESS_READY THEN
				step 							:= 30;
			ELSIF targetSlot.Shuttle.controlif = 0 THEN
				step 							:= 0;
			END_IF

		30:	(* Check Assemble Status and Slot Status *)
			IF (gSts.AsmState = E_ASM_PROCESS OR gSts.AsmState = E_ASM_IDLE)
				AND targetSlot.Interface = E_SLOT_PROCESS_READY THEN
				interface.Trak.ShuttleArrived	:= TRUE;
				fbShuttleOutCheck.Enable		:= TRUE;
				step 							:= 100;
			END_IF

		100: (* Wait Proess End and Next Stage Ready *)
			IF interface.Equipment.Done = TRUE AND NextReady THEN
				//Start to Read Data from PLC
				bBlockReadOnce					:= TRUE;
				step 							:= 101;
			END_IF

		101:
			IF bBlockReadOnceAck = TRUE THEN
				// Save Current Process Status
				userData.ProcessStatus			:= currentProcess;

				// Read process data from PLC
				brsmemcpy(ADR(userData.Data[0]), ADR(interface.Equipment.Data2[0]), SIZEOF(interface.Equipment.Data2));

				// End to Read Data from PLC
				bBlockReadOnce					:= FALSE;
				step := 110;
			END_IF

		110: 	//Write User Data
			fbUserData.DataAddress 				:= ADR(userData);
			fbUserData.DataSize 				:= SIZE_OF_USERDATA;
			fbUserData.Mode						:= mcACPTRAK_USERDATA_SET;
			fbUserData.Execute 					:= TRUE;

			IF fbUserData.Done = TRUE THEN
				fbUserData.Execute 				:= FALSE;
				//	interface.Trak.ShuttleArrived 	:= FALSE;
				targetSlot.Interface 			:= E_SLOT_TAKEOUT_READY;
				targetSlot.NextStage			:= nextSlot;
				step 							:= 120;
			END_IF

		120: 	//Done Check
			IF interface.Equipment.Done = FALSE THEN
				step 						:= 0;
			END_IF
	END_CASE;

	IF fbShuttleOutCheck.EventCount > 0 THEN
		interface.Trak.ShuttleArrived	:= FALSE;
		fbShuttleOutCheck.Enable		:= FALSE;
	END_IF

	IF targetSlot.Shuttle.controlif = 0 AND shuttleID <> '' THEN
		brsmemset(ADR(interface.Trak.Data[0]),0,11);
	END_IF

	fbUserData();
	fbShuttleOutCheck();
	Timer();
	Timer2();

END_PROGRAM
```

### Program Logical/Source/Control/ifStage18 (IEC) - Unloading

#### Main.st
```iecst
PROGRAM _INIT
	currentProcess							:= E_PROCESS_Stage18;
	fbUserData.Axis							:= ADR(StStage[17].Shuttle);
	nextSlot 								:= ADR(StStage[18]);

	fbShuttleOutCheck.ProcessPoint			:= ADR(ptStage18);

	targetSlot ACCESS ADR(StStage[17]);
	shuttleID ACCESS ADR(interface.Trak.Data[0]);
END_PROGRAM

PROGRAM _CYCLIC
	IF gSim = TRUE THEN
		bBlockReadOnceAck := bBlockReadOnce;
		bBlockSendOnceAck := bBlockSendOnce;
		bBlockSendShuttleIDAck := bBlockSendShuttleID;

		IF interface.Trak.ShuttleArrived = TRUE THEN
			interface.Equipment.Ready 		:= FALSE;

			tmr.IN 							:= TRUE;
			tmr.PT 							:= T#1s;
		END_IF

		IF tmr.Q = TRUE THEN
			interface.Equipment.Done 		:= TRUE;
		END_IF

		IF interface.Trak.ShuttleArrived = FALSE THEN
			tmr.IN							:= FALSE;
			interface.Equipment.Ready 		:= TRUE;
			interface.Equipment.Done 		:= FALSE;
		END_IF

		tmr();
	END_IF

	IF targetSlot.Interface = E_SLOT_UNKNOWN THEN
		step 				:= 0;
	END_IF

	CASE step OF
		0:	(* Modbus Interface Initialize and Shuttle Check *)
			bBlockSendShuttleID					:= FALSE;
			bBlockSendOnce						:= FALSE;
			bBlockReadOnce						:= FALSE;

			//interface.Trak.ShuttleArrived		:= FALSE;

			IF targetSlot.Shuttle.controlif <> 0 AND bBlockSendOnceAck = FALSE AND bBlockReadOnceAck = FALSE AND bBlockSendShuttleIDAck = FALSE THEN
				step 							:= 10;
			END_IF

		10:	(* Read Shuttle Data from userData *)
			fbUserData.DataAddress 				:= ADR(userData);
			fbUserData.DataSize 				:= SIZEOF(userData);
			fbUserData.Mode						:= mcACPTRAK_USERDATA_GET;
			fbUserData.Execute 					:= TRUE;

			IF fbUserData.Done = TRUE THEN
				//End to Read Data fron user Data
				fbUserData.Execute 				:= FALSE;

				//Copy User Data to Modbus IO
				brsmemcpy(ADR(interface.Trak.Data[0]),ADR(userData.SerialNumber), 11);
				brsmemcpy(ADR(interface.Trak.Data2[0]),ADR(userData.Data[0]), SIZEOF(userData.Data));

				//Start to Write userdata to Modbus
				bBlockSendOnce					:= TRUE;
				bBlockSendShuttleID				:= TRUE;
				step 							:= 11;
			END_IF

		11: (* Check End of write to Modbus *)
			IF bBlockSendOnceAck AND bBlockSendShuttleIDAck THEN
				bBlockSendOnce					:= FALSE;
				bBlockSendShuttleID				:= FALSE;
				step							:= 20;
			END_IF

		20: (* Check Process Ready *)
			IF targetSlot.Interface = E_SLOT_PROCESS_READY THEN
				step 							:= 30;
			ELSIF targetSlot.Shuttle.controlif = 0 THEN
				step 							:= 0;
			END_IF

		30:	(* Check Assemble Status and Slot Status *)
			IF (gSts.AsmState = E_ASM_PROCESS OR gSts.AsmState = E_ASM_IDLE)
				AND targetSlot.Interface = E_SLOT_PROCESS_READY THEN
				interface.Trak.ShuttleArrived	:= TRUE;
				fbShuttleOutCheck.Enable		:= TRUE;
				step 							:= 100;
			END_IF

		100: (* Wait Proess End and Next Stage Ready *)
			IF interface.Equipment.Done = TRUE AND NextReady THEN
				//Start to Read Data from PLC
				bBlockReadOnce					:= TRUE;
				step 							:= 101;
			END_IF

		101:
			IF bBlockReadOnceAck = TRUE THEN
				// Save Current Process Status
				userData.ProcessStatus			:= currentProcess;

				// Read process data from PLC
				brsmemcpy(ADR(userData.Data[0]), ADR(interface.Equipment.Data2[0]), SIZEOF(interface.Equipment.Data2));

				// End to Read Data from PLC
				bBlockReadOnce					:= FALSE;
				step := 110;
			END_IF

		110: 	//Write User Data
			fbUserData.DataAddress 				:= ADR(userData);
			fbUserData.DataSize 				:= SIZE_OF_USERDATA;
			fbUserData.Mode						:= mcACPTRAK_USERDATA_SET;
			fbUserData.Execute 					:= TRUE;

			IF fbUserData.Done = TRUE THEN
				fbUserData.Execute 				:= FALSE;
				//	interface.Trak.ShuttleArrived 	:= FALSE;
				targetSlot.Interface 			:= E_SLOT_TAKEOUT_READY;
				targetSlot.NextStage			:= nextSlot;
				step 							:= 120;
			END_IF

		120: 	//Done Check
			IF interface.Equipment.Done = FALSE THEN
				step 						:= 0;
			END_IF
	END_CASE;

	IF fbShuttleOutCheck.EventCount > 0 THEN
		interface.Trak.ShuttleArrived	:= FALSE;
		fbShuttleOutCheck.Enable		:= FALSE;
	END_IF

	IF targetSlot.Shuttle.controlif = 0 AND shuttleID <> '' THEN
		brsmemset(ADR(interface.Trak.Data[0]),0,11);
	END_IF

	fbUserData();
	fbShuttleOutCheck();
	Timer();
	Timer2();

END_PROGRAM
```

### Program Logical/Source/Control/ifStage19 (IEC) - Clean

#### Main.st
```iecst
PROGRAM _INIT
	currentProcess							:= E_PROCESS_Stage19;
	fbUserData.Axis							:= ADR(StStage[18].Shuttle);
//	nextSlot 								:= ADR(St_AnodeLoading);

	fbShuttleOutCheck.ProcessPoint			:= ADR(ptStage19);

	targetSlot ACCESS ADR(StStage[18]);
	shuttleID ACCESS ADR(interface.Trak.Data[0]);

	NextReady								:= TRUE;
END_PROGRAM

PROGRAM _CYCLIC
	IF gSim = TRUE THEN
		bBlockReadOnceAck := bBlockReadOnce;
		bBlockSendOnceAck := bBlockSendOnce;
		bBlockSendShuttleIDAck := bBlockSendShuttleID;

		IF interface.Trak.ShuttleArrived = TRUE THEN
			interface.Equipment.Ready 		:= FALSE;

			tmr.IN 							:= TRUE;
			tmr.PT 							:= T#1s;
		END_IF

		IF tmr.Q = TRUE THEN
			interface.Equipment.Done 		:= TRUE;
		END_IF

		IF interface.Trak.ShuttleArrived = FALSE THEN
			tmr.IN							:= FALSE;
			interface.Equipment.Ready 		:= TRUE;
			interface.Equipment.Done 		:= FALSE;
		END_IF

		tmr();
	END_IF

	IF targetSlot.Interface = E_SLOT_UNKNOWN THEN
		step 				:= 0;
	END_IF

	CASE step OF
		0:	(* Modbus Interface Initialize and Shuttle Check *)
			bBlockSendShuttleID					:= FALSE;
			bBlockSendOnce						:= FALSE;
			bBlockReadOnce						:= FALSE;

			//interface.Trak.ShuttleArrived		:= FALSE;

			IF targetSlot.Shuttle.controlif <> 0 AND bBlockSendOnceAck = FALSE AND bBlockReadOnceAck = FALSE AND bBlockSendShuttleIDAck = FALSE THEN
				step 							:= 10;
			END_IF

		10:	(* Read Shuttle Data from userData *)
			fbUserData.DataAddress 				:= ADR(userData);
			fbUserData.DataSize 				:= SIZEOF(userData);
			fbUserData.Mode						:= mcACPTRAK_USERDATA_GET;
			fbUserData.Execute 					:= TRUE;

			IF fbUserData.Done = TRUE THEN
				//End to Read Data fron user Data
				fbUserData.Execute 				:= FALSE;

				//Copy User Data to Modbus IO
				brsmemcpy(ADR(interface.Trak.Data[0]),ADR(userData.SerialNumber), 11);
				brsmemcpy(ADR(interface.Trak.Data2[0]),ADR(userData.Data[0]), SIZEOF(userData.Data));

				//Start to Write userdata to Modbus
				bBlockSendOnce					:= TRUE;
				bBlockSendShuttleID				:= TRUE;
				step 							:= 11;
			END_IF

		11: (* Check End of write to Modbus *)
			IF bBlockSendOnceAck AND bBlockSendShuttleIDAck THEN
				bBlockSendOnce					:= FALSE;
				bBlockSendShuttleID				:= FALSE;
				step							:= 20;
			END_IF

		20: (* Check Process Ready *)
			IF targetSlot.Interface = E_SLOT_PROCESS_READY THEN
				step 							:= 30;
			ELSIF targetSlot.Shuttle.controlif = 0 THEN
				step 							:= 0;
			END_IF

		30:	(* Check Assemble Status and Slot Status *)
			IF (gSts.AsmState = E_ASM_PROCESS OR gSts.AsmState = E_ASM_IDLE)
				AND targetSlot.Interface = E_SLOT_PROCESS_READY THEN
				interface.Trak.ShuttleArrived	:= TRUE;
				fbShuttleOutCheck.Enable		:= TRUE;
				step 							:= 100;
			END_IF

		100: (* Wait Proess End and Next Stage Ready *)
			IF interface.Equipment.Done = TRUE AND NextReady THEN
				//Start to Read Data from PLC
				bBlockReadOnce					:= TRUE;
				step 							:= 101;
			END_IF

		101:
			IF bBlockReadOnceAck = TRUE THEN
				// Save Current Process Status
				userData.ProcessStatus			:= currentProcess;

				// Read process data from PLC
				brsmemcpy(ADR(userData.Data[0]), ADR(interface.Equipment.Data2[0]), SIZEOF(interface.Equipment.Data2));

				// End to Read Data from PLC
				bBlockReadOnce					:= FALSE;
				step := 110;
			END_IF

		110: 	//Write User Data
			fbUserData.DataAddress 				:= ADR(userData);
			fbUserData.DataSize 				:= SIZE_OF_USERDATA;
			fbUserData.Mode						:= mcACPTRAK_USERDATA_SET;
			fbUserData.Execute 					:= TRUE;

			IF fbUserData.Done = TRUE THEN
				fbUserData.Execute 				:= FALSE;
				//	interface.Trak.ShuttleArrived 	:= FALSE;
				targetSlot.Interface 			:= E_SLOT_TAKEOUT_READY;
				targetSlot.NextStage			:= nextSlot;
				step 							:= 120;
			END_IF

		120: 	//Done Check
			IF interface.Equipment.Done = FALSE THEN
				step 						:= 0;
			END_IF
	END_CASE;

	IF fbShuttleOutCheck.EventCount > 0 THEN
		interface.Trak.ShuttleArrived	:= FALSE;
		fbShuttleOutCheck.Enable		:= FALSE;
	END_IF

	IF targetSlot.Shuttle.controlif = 0 AND shuttleID <> '' THEN
		brsmemset(ADR(interface.Trak.Data[0]),0,11);
	END_IF

	fbUserData();
	fbShuttleOutCheck();
	Timer();
	Timer2();

END_PROGRAM
```

### VisionVariables.var
```iecst
(*-----------------------------------------------------------------------------------------------------------------------------------------*)
(*Global variables for sensor hardware and vision functions*)
VAR
	gCodeReader : typCodeReaderMain; (*Data that is specific for the code reader*)
	gVisionSensor : typVisionMain; (*General vision functions that are independent from the inspection function*)
	NettimeCurrent_us : DINT; (*Current Powerlink nettime*)
END_VAR
VAR RETAIN
	gParVision : recVariable; (*Structure that contains the recipe variables*)
END_VAR
(*-----------------------------------------------------------------------------------------------------------------------------------------*)
(*Global constants*)
VAR CONSTANT
	MAX_NUM_CAMS : UINT := 6; (*Maximum number of camera's*)
	MAX_NUM_RESULTS : UINT := 10; (*Maximum number of results*)
	MAX_NUM_PRODUCTS : UINT := 8; (*Maximum number of products for color detection*)
	MAX_IDX_VA_LIST : UINT := 19; (*Maximum number of entrys in the Vision Application list*)
	DEVICE_NAME : STRING[40] := 'VisionFileDevice'; (*File device where the images and recipes are stored*)
	NETTIME_DEFAULT_DELAY : UDINT := 30000; (*This delay is used when software trigger is used and nettime is enabled*)
	NETTIME_ENABLE : BOOL := FALSE; (*Enable nettime code, this generates the nettime when using manual triggers*)
	MAX_NUM_CODETYPES : USINT := 69; (*Maximum number of code types*)
END_VAR
VAR
	CodeTypes : {REDUND_UNREPLICABLE} ARRAY[0..MAX_NUM_CODETYPES] OF STRING[80] := ['Auto Identify (0)','2/5 Industrial (1)','2/5 Interleaved (2)','Codebar (3)','Code 32 (4)','Code 39 (5)','Code 93 (6)','Code 128 (7)','MSI (8)','PharmaCode (9)','EAN-8 (10)','EAN-8 Add-On 2 (11)','EAN-8 Add-On 5 (12)','EAN-13 (13)','EAN-13 Add-On 2 (14)','EAN-13 Add-On 5 (15)',4(''),'UPC-A (20)','UPC-A Add-On 2 (21)','UPC-A Add-On 5 (22)','UPC-E (23)','UPC-E Add-On 2 (24)','UPC-E Add-On 5 (25)',4(''),'GS1-128 (30)','GS1 DataBar Omnidirectional (31)','GS1 DataBar Truncated (32)','GS1 DataBar Stacked (33)','GS1 DataBar Stacked Omnidirectional (34)','GS1 DataBar Limited (35)','GS1 DataBar Expanded (36)','GS1 DataBar ExpandedStacked (37)',12(''),'Data Matrix ECC200 (50)','QR Code Model 1 (51)','QR Code Model 2 (52)','Micro QRCode (53)','PDF417 (54)','Aztec Code (55)',4(''),'GS1 Data Matrix (60)','GS1 QR Code Model 1 (61)','GS1 QR Code Model 2 (62)','GS1 Aztec Code (63)',6('')]; (*Codes types for code reading*)
	gBarCodeReader : VisionInterface_typ;
END_VAR
```

### VisionTypes.typ
```iecst
(*-----------------------------------------------------------------------------------------------------------------------------------------*)
(*General vision structures*)

TYPE
	typVisionMain : 	STRUCT
		CMD : typVisionCommand;
		CFG : typVisionConfig;
		DAT : typVisionData;
		FCT : typVisionFunction;
		DIA : typVisionDiag;
		OPT : typVisionOptics;
		HW : typVisionHW;
	END_STRUCT;
	typVisionCommand : 	STRUCT
		ImageTrigger : BOOL;
		ImageTriggerReset : BOOL;
		AutoSetupStartStop : BOOL;
		VaSwitchApplication : BOOL;
		SaveDiagData : BOOL;
		ReadCameraInfo : BOOL;
	END_STRUCT;
	typVisionConfig : 	STRUCT
		VisionFunction : enumVisionFunction;
		PowerlinkNode : USINT;
		DataStructure : UDINT;
		ComponentLink : ViComponentType;
		ResolutionWidth_X : UINT; (*Nr of sensor pixels in x direction (width). Is always bigger than height*)
		ResolutionHeight_Y : UINT; (*Nr of sensor pixels in y direction (height). Is always smaller than width*)
	END_STRUCT;
	typVisionFunction : 	STRUCT
		ApplicationName : STRING[40];
		Status : DINT;
	END_STRUCT;
	typVisionDiag : 	STRUCT
		DiagName : STRING[80] := 'diag.tgz';
		Status : DINT;
	END_STRUCT;
	typVisionData : 	STRUCT
		Enable : BOOL := FALSE;
		MaxItemCnt : USINT := 1;
		NettimeDelay : DINT;
		Timeout : UINT := 500;
		Gain : USINT := 1;
		Focus : UINT := 15951;
		Exposure : UDINT := 11;
		FlashColor : USINT := 1;
		FlashSegment : USINT := 15;
		LedColor : USINT;
		IRFilter : BOOL;
		OffsetROIX : DINT;
		OffsetROIY : DINT;
		OffsetROIRotationCenterX : DINT;
		OffsetROIRotationCenterY : DINT;
		OffsetROIOrientation : INT;
		ChromaticLock : BOOL;
		Alignment : USINT;
		AutoSetupGain : USINT;
		AutoSetupFocus : UINT;
		AutoSetupExposure : UDINT;
		AcquisitionAcceptedCnt : USINT;
		AcquisitionCompletedCnt : USINT;
		AcquisitionFailedCnt : USINT;
		LightWarningCnt : USINT;
		ImageProcessingError : UINT;
		ImageProcessingActive : BOOL;
		ImageNettime : DINT;
		ProcessingTimeCamera : UINT;
		ProcessingTimeFunction : UINT;
		ResultCnt : USINT;
		CockpitIsActive : BOOL;
		Status : UDINT;
		StatusText : STRING[30];
		Active : BOOL;
	END_STRUCT;
	typVisionHW : 	STRUCT
		Connected : BOOL;
		Ready : BOOL;
		DigitalInput01 : BOOL;
		DigitalOutput01 : BOOL;
		DigitalOutputStatus01 : BOOL;
		DigitalOutput02 : BOOL;
		DigitalOutputStatus02 : BOOL;
		SerialNumber : UDINT;
		ID : UDINT;
		Variant : UDINT;
		Firmware : UDINT;
		Undervoltage : BOOL;
		Temperature : SINT;
	END_STRUCT;
	typVisionOptics : 	STRUCT
		OrderNr : STRING[40];
		Binning : BOOL;
		ResolutionX : INT;
		ResolutionY : INT;
		Lens : USINT;
		Sensor : USINT;
		ValidDistance : BOOL;
		Distance_mm : LREAL;
		DistanceLens_mm : LREAL;
		HyperFocalDistance_mm : LREAL;
		PixelSize_um : LREAL;
		PixelSizeBinning_um : LREAL;
		FocalLength_mm : LREAL;
		MinObjectDist_mm : LREAL;
		MaxObjectDist_mm : LREAL;
		Aperture : LREAL;
		CircleOfConfusion_mm : LREAL;
		DepthOfFieldNearPos_mm : LREAL;
		DepthOfFieldFarPos_mm : LREAL;
		DepthOfField_mm : LREAL;
		FieldOfView_X_mm : LREAL;
		FieldOfView_Y_mm : LREAL;
		Resolution_mmPerPx : LREAL;
	END_STRUCT;
	enumVisionFunction :
		(
		enumFunctionNone,
		enumBlob,
		enumCoderReader,
		enumMatch,
		enumMeasurement,
		enumOCR,
		enumPixelCounter
		);
END_TYPE

(*-----------------------------------------------------------------------------------------------------------------------------------------*)
(*Vision specific structures*)

TYPE
	typCodeReaderMain : 	STRUCT  (*Code reader structures*)
		CodeType : USINT := 50;
		GradingEnable : BOOL;
		RobustnessEnable : BOOL;
		ParameterMode : USINT := 0;
		ParameterOptimization : USINT;
		BarcodeText : ARRAY[1..MAX_NUM_RESULTS]OF STRING[100];
		BarcodeType : ARRAY[1..MAX_NUM_RESULTS]OF USINT;
		PositionX : ARRAY[1..MAX_NUM_RESULTS]OF DINT;
		PositionY : ARRAY[1..MAX_NUM_RESULTS]OF DINT;
		Orientation : ARRAY[1..MAX_NUM_RESULTS]OF INT;
		Grading : ARRAY[1..MAX_NUM_RESULTS]OF SINT;
		EnhancedGrading : ARRAY[1..23]OF USINT;
	END_STRUCT;
END_TYPE

(*------------------------------------------------------------------------------------------------------------------------------------------------------------------------------------------------------------------------*)
(*Structure that contains the recipe variables*)

TYPE
	recVariable : 	STRUCT
		Cam : recVariableCam;
	END_STRUCT;
	recVariableCam : 	STRUCT
		ApplicationName : STRING[40];
		MaxItemCnt : USINT; (*Default 1*)
		Timeout : UINT; (*Default 200*)
		Gain : USINT;
		Focus : UINT;
		Exposure : UDINT;
		FlashColor : USINT; (*Default is 1*)
		FlashSegment : USINT; (*Default is 15*)
	END_STRUCT;
END_TYPE

(*------------------------------------------------------------------------------------------------------------------------------------------------------------------------------------------------------------------------*)
(*Structure that contains the recipe variables*)

TYPE
	VisionInterface_typ : 	STRUCT
		Enable : BOOL;
		Trigger : BOOL;
		TakeCount : USINT;
		SerialNumber : STRING[100];
	END_STRUCT;
END_TYPE
```

### Program Logical/Source/Vision/Vi_main (IEC)

#### Vi_main.st - Init, cyclic, exit code
```iecst
// --------------------------------------------------------------------------------------------------------------------
// General vision task. This is a support task for the mappVision. The following functions are implemneted
// - Translate some values in text messages
// - Reset camera trigger when inspection is finsihed
// - Load vision application
// - Save diagnostic data
// Version 2.x (Check revision history for details)
// --------------------------------------------------------------------------------------------------------------------
PROGRAM _INIT
	gVisionSensor;
	gCodeReader;
END_PROGRAM

// -----------------------------------------------------------------------------------------------------------
// Cyclic part
// -----------------------------------------------------------------------------------------------------------
PROGRAM _CYCLIC
	// -----------------------------------------------------------------------------------------------------------
	// Translate camera status in readable text
	// -----------------------------------------------------------------------------------------------------------
	IF gVisionSensor.DAT.Status = 0 THEN // Display only a single 0
		gVisionSensor.DAT.StatusText := 'Ready';
	ELSIF gVisionSensor.DAT.Status = 16#00000001 THEN
		gVisionSensor.DAT.StatusText := 'Image acquisition';
	ELSIF gVisionSensor.DAT.Status = 16#00000002 THEN
		gVisionSensor.DAT.StatusText := 'Waiting trigger';
	ELSIF gVisionSensor.DAT.Status = 16#00000010 THEN
		gVisionSensor.DAT.StatusText := 'Searching settings';
	ELSIF gVisionSensor.DAT.Status = 16#00000080 THEN
		gVisionSensor.DAT.StatusText := 'Setting focus';
	ELSIF gVisionSensor.DAT.Status = 16#00000090 THEN
		gVisionSensor.DAT.StatusText := 'Searching settings';
	ELSIF gVisionSensor.DAT.Status = 16#00000800 THEN
		gVisionSensor.DAT.StatusText := 'Cam CPU not ready';
	ELSIF gVisionSensor.DAT.Status = 16#00001000 THEN
		gVisionSensor.DAT.StatusText := 'Cam sensor not ready';
	ELSIF gVisionSensor.DAT.Status = 16#01000000 OR gVisionSensor.DAT.Status = 16#02000000 OR gVisionSensor.DAT.Status = 16#03000000 THEN
		gVisionSensor.DAT.StatusText := 'OS check/update';
	ELSIF gVisionSensor.DAT.Status = 16#80000000 THEN
		gVisionSensor.DAT.StatusText := 'Vision cockpit active';
	ELSE
		// Display the status in hex format 0x02000800
		gVisionSensor.DAT.StatusText := '';
		FOR i := 0 TO 28 BY 4 DO
			gVisionSensor.DAT.StatusText := CONCAT(MID(HexTab, 1, LIMIT(1, UDINT_TO_INT((SHR(gVisionSensor.DAT.Status, i) AND 16#0000000F) + 1), 16)), gVisionSensor.DAT.StatusText);
		END_FOR
		gVisionSensor.DAT.StatusText := CONCAT('0x', gVisionSensor.DAT.StatusText);
	END_IF

	// -----------------------------------------------------------------------------------------------------------
	// Check if vision cockpit is open
	// -----------------------------------------------------------------------------------------------------------
	gVisionSensor.DAT.CockpitIsActive := (gVisionSensor.DAT.Status AND 16#8000_0000) > 0;

	// -----------------------------------------------------------------------------------------------------------
	// Auto setup handling
	// -----------------------------------------------------------------------------------------------------------
	IF(gVisionSensor.CMD.AutoSetupStartStop AND gVisionSensor.DAT.Status <> 0) THEN
		AutoSetupRunning := TRUE;
	ELSIF NOT gVisionSensor.CMD.AutoSetupStartStop THEN
		AutoSetupRunning := FALSE;
	END_IF
	IF(gVisionSensor.CMD.AutoSetupStartStop AND gVisionSensor.DAT.Status = 0 AND AutoSetupRunning) THEN // Setup successfully finished
		gVisionSensor.DAT.Gain					:= gVisionSensor.DAT.AutoSetupGain;
		gVisionSensor.DAT.Focus					:= gVisionSensor.DAT.AutoSetupFocus;
		gVisionSensor.DAT.Exposure				:= gVisionSensor.DAT.AutoSetupExposure;
		gVisionSensor.CMD.AutoSetupStartStop	:= FALSE;
		AutoSetupRunning						:= FALSE;
		TON_DelayAfterAutoSetup.IN				:= TRUE;
	END_IF
	TON_DelayAfterAutoSetup(PT := T#50ms);
	IF TON_DelayAfterAutoSetup.Q THEN // After the camera tells it is ready, we need to wait still at least ca 20ms, otherwise it does not accept the trigger
		TON_DelayAfterAutoSetup.IN := FALSE;
		IF gVisionSensor.HW.Ready AND NOT gVisionSensor.DAT.ImageProcessingActive THEN
			IF NETTIME_ENABLE THEN
				gVisionSensor.DAT.NettimeDelay := NettimeCurrent_us + NETTIME_DEFAULT_DELAY;
			END_IF
			gVisionSensor.CMD.ImageTrigger	:= TRUE;
			gVisionSensor.DAT.Active		:= TRUE;
		END_IF
	END_IF

	// -----------------------------------------------------------------------------------------------------------
	// Reset image trigger, reload web page and store image when process is finished
	// -----------------------------------------------------------------------------------------------------------
	IF ((gVisionSensor.DAT.AcquisitionCompletedCnt <> AcquisitionCompletedCntOld OR gVisionSensor.DAT.AcquisitionFailedCnt <> AcquisitionFailedCntOld) AND NOT gVisionSensor.DAT.ImageProcessingActive AND gVisionSensor.HW.Ready) THEN
		AcquisitionCompletedCntOld		:= gVisionSensor.DAT.AcquisitionCompletedCnt;
		AcquisitionFailedCntOld			:= gVisionSensor.DAT.AcquisitionFailedCnt;
		gVisionSensor.CMD.ImageTrigger	:= FALSE;
		gVisionSensor.DAT.Active		:= FALSE;
	END_IF

	// -----------------------------------------------------------------------------------------------------------
	// Reset trigger when timed out
	// -----------------------------------------------------------------------------------------------------------
	IF gVisionSensor.CMD.ImageTrigger THEN
		TriggerTimeoutSensor.IN := TRUE;
		TriggerTimeoutSensor.PT := REAL_TO_TIME(gVisionSensor.DAT.Timeout * 1.25);
		IF TriggerTimeoutSensor.Q THEN
			gVisionSensor.CMD.ImageTrigger			:= FALSE;
			gVisionSensor.CMD.ImageTriggerReset		:= TRUE;
			gVisionSensor.DAT.Active				:= FALSE;
		END_IF
	ELSE
		TriggerTimeoutSensor.IN := FALSE;
		gVisionSensor.CMD.ImageTriggerReset := FALSE;
	END_IF
	TriggerTimeoutSensor();

	// -----------------------------------------------------------------------------------------------------------
	// Load vision application
	// -----------------------------------------------------------------------------------------------------------
	IF (gVisionSensor.CMD.VaSwitchApplication) THEN
		ViBaseLoadApplication_01.MpLink	:= ADR(gVisionSensor.CFG.ComponentLink);
		ViBaseLoadApplication_01.Name	:= ADR(gVisionSensor.FCT.ApplicationName);
		gVisionSensor.FCT.Status := ERR_FUB_BUSY;

		// -----------------------------------------------------------------------------------------------------------
		// OK
		IF (ViBaseLoadApplication_01.Done) THEN
			gVisionSensor.FCT.Status := ERR_OK;
			gVisionSensor.CMD.VaSwitchApplication := FALSE;
			// -----------------------------------------------------------------------------------------------------------
			// Error
		ELSIF (NOT ViBaseLoadApplication_01.Busy AND ViBaseLoadApplication_01.Error) THEN
			gVisionSensor.FCT.Status := ViBaseLoadApplication_01.StatusID;
			gVisionSensor.CMD.VaSwitchApplication := FALSE;
		END_IF
	END_IF
	ViBaseLoadApplication_01.Execute := gVisionSensor.CMD.VaSwitchApplication;
	ViBaseLoadApplication_01();
	// Dont proceed until loading is finished
	IF (gVisionSensor.CMD.VaSwitchApplication) THEN
		RETURN;
	END_IF

	// -----------------------------------------------------------------------------------------------------------
	// Save diagnostic data
	// -----------------------------------------------------------------------------------------------------------
	IF (gVisionSensor.CMD.SaveDiagData) THEN
		// Delete old file first
		FDelete.enable := gVisionSensor.CMD.SaveDiagData AND NOT ViBaseSaveDiagData_01.Execute;
		FDelete.pDevice := ADR(DEVICE_NAME);
		FDelete.pName := ADR(gVisionSensor.DIA.DiagName);
		IF (FDelete.status <> ERR_FUB_BUSY) THEN
			ViBaseSaveDiagData_01.Execute := TRUE;
		END_IF
		// Upload diagnostic information
		ViBaseSaveDiagData_01.MpLink := ADR(gVisionSensor.CFG.ComponentLink);
		ViBaseSaveDiagData_01.DeviceName := ADR(DEVICE_NAME);
		ViBaseSaveDiagData_01.FileName := ADR(gVisionSensor.DIA.DiagName);
		gVisionSensor.DIA.Status := ERR_FUB_BUSY;

		// -----------------------------------------------------------------------------------------------------------
		// OK
		IF (ViBaseSaveDiagData_01.Done) THEN
			gVisionSensor.DIA.Status := ERR_OK;
			ViBaseSaveDiagData_01.Execute := FALSE;
			gVisionSensor.CMD.SaveDiagData := FALSE;
			// -----------------------------------------------------------------------------------------------------------
			// Error
		ELSIF (NOT ViBaseSaveDiagData_01.Busy AND ViBaseSaveDiagData_01.Error) THEN
			gVisionSensor.DIA.Status := ViBaseSaveDiagData_01.StatusID;
			ViBaseSaveDiagData_01.Execute := FALSE;
			gVisionSensor.CMD.SaveDiagData := FALSE;
		END_IF
	END_IF
	ViBaseSaveDiagData_01();
	FDelete();
	// Dont proceed until loading is finished
	IF (gVisionSensor.CMD.SaveDiagData) THEN
		RETURN;
	END_IF

	// -----------------------------------------------------------------------------------------------------------
	// Read camera info
	// -----------------------------------------------------------------------------------------------------------
	CASE OpticsReadStep[idSensor] OF
		// -----------------------------------------------------------------------------------------------------------
		// Wait
		0:
			IF gVisionSensor.CMD.ReadCameraInfo THEN
				gVisionSensor.OPT.OrderNr	:= '';
				Index := 0;
				OpticsReadStep[idSensor]	:= 1;
			END_IF
			// -----------------------------------------------------------------------------------------------------------
			// Create DiagInformation
		1:
			DiagCreateInfo_0.enable			:= TRUE;
			DiagCreateInfo_0.infoKind		:= asdiagPLUGGED;
			DiagCreateInfo_0();
			IF DiagCreateInfo_0.status = 0 THEN
				OpticsReadStep[idSensor] := 2;
			ELSIF DiagCreateInfo_0.status <> ERR_FUB_BUSY THEN
				OpticsReadStep[idSensor] := 90;
			END_IF
			// -----------------------------------------------------------------------------------------------------------
			// Read HW-ID and compare with selected camera
		2:
			DiagGetNumInfo_0.enable			:= TRUE;
			DiagGetNumInfo_0.ident			:= DiagCreateInfo_0.ident;
			DiagGetNumInfo_0.index			:= Index;
			DiagGetNumInfo_0.infoCode		:= asdiagPLUGGED_MODNO;
			DiagGetNumInfo_0();
			IF DiagGetNumInfo_0.status = 0 THEN
				//IF DiagGetNumInfo_0.value = gVisionSensor[visSelectedSensor].HW.ID THEN
				IF DiagGetNumInfo_0.value = gVisionSensor.HW.ID THEN
					OpticsReadStep[idSensor] := 3;
				ELSE
					Index := Index + 1;
					IF Index >= DiagCreateInfo_0.nrEntries THEN
						OpticsReadStep[idSensor] := 91;
					END_IF
				END_IF
			ELSIF DiagGetNumInfo_0.status <> ERR_FUB_BUSY THEN
				OpticsReadStep[idSensor] := 92;
			END_IF
			// -----------------------------------------------------------------------------------------------------------
			// Read ordernumber
		3:
			DiagGetStrInfo_0.enable			:= TRUE;
			DiagGetStrInfo_0.ident			:= DiagCreateInfo_0.ident;
			DiagGetStrInfo_0.index			:= Index;
			DiagGetStrInfo_0.infoCode		:= asdiagPLUGGED_MODULE;
			DiagGetStrInfo_0.pBuffer		:= ADR(gVisionSensor.OPT.OrderNr);
			DiagGetStrInfo_0.bufferLen		:= SIZEOF(gVisionSensor.OPT.OrderNr) - 1;
			DiagGetStrInfo_0();
			IF DiagGetStrInfo_0.status = 0 THEN
				OpticsReadStep[idSensor] := 10;
			ELSIF DiagGetStrInfo_0.status <> ERR_FUB_BUSY THEN
				OpticsReadStep[idSensor] := 93;
			END_IF
			// -----------------------------------------------------------------------------------------------------------
			// Release info function block
		10:
			DiagDisposeInfo_0.enable		:= TRUE;
			DiagDisposeInfo_0.ident			:= DiagCreateInfo_0.ident;
			DiagDisposeInfo_0();
			IF DiagDisposeInfo_0.status = 0 THEN
				OpticsReadStep[idSensor] := 20;
			ELSIF DiagDisposeInfo_0.status <> ERR_FUB_BUSY THEN
				OpticsReadStep[idSensor] := 94;
			END_IF
			// -----------------------------------------------------------------------------------------------------------
			// Get the info to the actual camara
		20:
			IF brsstrlen(ADR(gVisionSensor.OPT.OrderNr)) = 18 THEN
				pChar ACCESS ADR(gVisionSensor.OPT.OrderNr) + 8; 	// Letter for Sensor
				CASE pChar OF
					16#31:  gVisionSensor.OPT.Sensor := SENSOR_1_3_MP; // ASCII '1'
					16#32:  gVisionSensor.OPT.Sensor := SENSOR_1_3_MP; // ASCII '2'
					16#34:  gVisionSensor.OPT.Sensor := SENSOR_3_5_MP; // ASCII '4'
					16#35:  gVisionSensor.OPT.Sensor := SENSOR_5_3_MP; // ASCII '5'
					ELSE
						OpticsReadStep[idSensor] := 95;
				END_CASE
				pChar ACCESS ADR(gVisionSensor.OPT.OrderNr) + 10; // first letter for optics (0 or M)
				CASE pChar OF
					16#30:  gVisionSensor.OPT.Lens := LENS_4_6; // ASCII '0'
					16#4D:  gVisionSensor.OPT.Lens := LENS_12_0_MACRO; // ASCII 'M'
					ELSE
						OpticsReadStep[idSensor] := 96;
				END_CASE
				pChar ACCESS ADR(gVisionSensor.OPT.OrderNr) + 11; // second letter for optics
				CASE pChar OF
					16#30:  gVisionSensor.OPT.Lens := LENS_4_6; // ASCII '0' // no optics
					16#32:  gVisionSensor.OPT.Lens := LENS_4_6; // ASCII '2'
					16#33:  gVisionSensor.OPT.Lens := LENS_6_0; // ASCII '3'
					16#34:  gVisionSensor.OPT.Lens := LENS_8_0; // ASCII '4'
					16#35: // ASCII '5'
					IF gVisionSensor.OPT.Lens = LENS_12_0_MACRO THEN
						// do noting, already selected
					ELSE
						gVisionSensor.OPT.Lens := LENS_12_0;
					END_IF
					16#36:  gVisionSensor.OPT.Lens := LENS_16_0; // ASCII '6'
					16#37:  gVisionSensor.OPT.Lens := LENS_25_0; // ASCII '7'
					ELSE
						OpticsReadStep[idSensor] := 97;
				END_CASE
				gVisionSensor.OPT.Distance_mm := gVisionSensor.DAT.Focus/100;
				gVisionSensor.CMD.ReadCameraInfo := FALSE;
				OpticsReadStep[idSensor] := 0;
			ELSE
				OpticsReadStep[idSensor] := 98;
			END_IF
		90..99: // auto reset errors
			gVisionSensor.CMD.ReadCameraInfo := FALSE;
			OpticsReadStep[idSensor] := 0;
	END_CASE

	// -----------------------------------------------------------------------------------------------------------
	// Set sensor parameter
	CASE gVisionSensor.OPT.Sensor OF
		SENSOR_1_3_MP:
			gVisionSensor.OPT.PixelSize_um		:= 4.8;
			gVisionSensor.OPT.ResolutionX		:= 1280;
			gVisionSensor.OPT.ResolutionY		:= 1024;
		SENSOR_3_5_MP:
			gVisionSensor.OPT.PixelSize_um		:= 3.2;
			gVisionSensor.OPT.ResolutionX		:= 2112;
			gVisionSensor.OPT.ResolutionY		:= 1664;
		SENSOR_5_3_MP:
			gVisionSensor.OPT.PixelSize_um		:= 3.2;
			gVisionSensor.OPT.ResolutionX		:= 2592;
			gVisionSensor.OPT.ResolutionY		:= 2048;
	END_CASE

	// -----------------------------------------------------------------------------------------------------------
	// Set lens parameter
	CASE gVisionSensor.OPT.Lens OF
		LENS_4_6:
			gVisionSensor.OPT.FocalLength_mm	:= 4.6;
			gVisionSensor.OPT.MinObjectDist_mm	:= 25;
			gVisionSensor.OPT.MaxObjectDist_mm	:= 65550;
			gVisionSensor.OPT.Aperture			:= 3.5;
		LENS_6_0:
			gVisionSensor.OPT.FocalLength_mm	:= 6.0;
			gVisionSensor.OPT.MinObjectDist_mm	:= 50;
			gVisionSensor.OPT.MaxObjectDist_mm	:= 65550;
			gVisionSensor.OPT.Aperture			:= 3.5;
		LENS_8_0:
			gVisionSensor.OPT.FocalLength_mm	:= 8.0;
			gVisionSensor.OPT.MinObjectDist_mm	:= 50;
			gVisionSensor.OPT.MaxObjectDist_mm	:= 65500;
			gVisionSensor.OPT.Aperture			:= 3.5;
		LENS_12_0:
			gVisionSensor.OPT.FocalLength_mm	:= 12.0;
			gVisionSensor.OPT.MinObjectDist_mm	:= 75;
			gVisionSensor.OPT.MaxObjectDist_mm	:= 5000;
			gVisionSensor.OPT.Aperture			:= 4.0;
		LENS_16_0:
			gVisionSensor.OPT.FocalLength_mm	:= 16.0;
			gVisionSensor.OPT.MinObjectDist_mm	:= 100;
			gVisionSensor.OPT.MaxObjectDist_mm	:= 1500;
			gVisionSensor.OPT.Aperture			:= 4.0;
		LENS_25_0:
			gVisionSensor.OPT.FocalLength_mm	:= 25.0;
			gVisionSensor.OPT.MinObjectDist_mm	:= 250;
			gVisionSensor.OPT.MaxObjectDist_mm	:= 1500;
			gVisionSensor.OPT.Aperture			:= 4.0;
		LENS_12_0_MACRO:
			gVisionSensor.OPT.FocalLength_mm	:= 12.0;
			gVisionSensor.OPT.MinObjectDist_mm	:= 35;
			gVisionSensor.OPT.MaxObjectDist_mm	:= 65;
			gVisionSensor.OPT.Aperture			:= 4.0;
	END_CASE
	gVisionSensor.OPT.ValidDistance := gVisionSensor.OPT.Distance_mm >= gVisionSensor.OPT.MinObjectDist_mm AND gVisionSensor.OPT.Distance_mm <= gVisionSensor.OPT.MaxObjectDist_mm;
	IF gVisionSensor.OPT.ValidDistance THEN
		gVisionSensor.OPT.DistanceLens_mm				:= gVisionSensor.OPT.Distance_mm + DISTANCE_FRONTGLASS_LENS_MM; // The lens is 15mm behind the front glass
		IF gVisionSensor.OPT.Binning THEN
			gVisionSensor.OPT.PixelSizeBinning_um		:= gVisionSensor.OPT.PixelSize_um * 2;
		ELSE
			gVisionSensor.OPT.PixelSizeBinning_um		:= gVisionSensor.OPT.PixelSize_um * 1;
		END_IF
		gVisionSensor.OPT.CircleOfConfusion_mm			:= gVisionSensor.OPT.PixelSizeBinning_um * 1 * SQRT(2.0) / 1000.0;
		gVisionSensor.OPT.HyperFocalDistance_mm			:= (gVisionSensor.OPT.FocalLength_mm * gVisionSensor.OPT.FocalLength_mm) / (gVisionSensor.OPT.Aperture * gVisionSensor.OPT.CircleOfConfusion_mm) + gVisionSensor.OPT.FocalLength_mm;
		gVisionSensor.OPT.DepthOfFieldNearPos_mm		:= gVisionSensor.OPT.DistanceLens_mm * (gVisionSensor.OPT.HyperFocalDistance_mm - gVisionSensor.OPT.FocalLength_mm) / (gVisionSensor.OPT.HyperFocalDistance_mm + gVisionSensor.OPT.DistanceLens_mm - 2 * gVisionSensor.OPT.FocalLength_mm) - DISTANCE_FRONTGLASS_LENS_MM;
		IF gVisionSensor.OPT.DistanceLens_mm < gVisionSensor.OPT.HyperFocalDistance_mm THEN
			gVisionSensor.OPT.DepthOfFieldFarPos_mm	:= gVisionSensor.OPT.DistanceLens_mm * (gVisionSensor.OPT.HyperFocalDistance_mm - gVisionSensor.OPT.FocalLength_mm) / (gVisionSensor.OPT.HyperFocalDistance_mm - gVisionSensor.OPT.DistanceLens_mm) - DISTANCE_FRONTGLASS_LENS_MM;
			gVisionSensor.OPT.DepthOfField_mm			:= gVisionSensor.OPT.DepthOfFieldFarPos_mm - gVisionSensor.OPT.DepthOfFieldNearPos_mm;
		ELSE
			gVisionSensor.OPT.DepthOfFieldFarPos_mm		:= -1; // Means "infinite"
			gVisionSensor.OPT.DepthOfField_mm			:= -1; // Means "infinite"
		END_IF
		gVisionSensor.OPT.FieldOfView_X_mm			:= gVisionSensor.OPT.PixelSizeBinning_um / 1000 * gVisionSensor.OPT.ResolutionX *(gVisionSensor.OPT.DistanceLens_mm / gVisionSensor.OPT.FocalLength_mm - 1.0);
		gVisionSensor.OPT.FieldOfView_Y_mm			:= gVisionSensor.OPT.PixelSizeBinning_um / 1000 * gVisionSensor.OPT.ResolutionY *(gVisionSensor.OPT.DistanceLens_mm / gVisionSensor.OPT.FocalLength_mm - 1.0);
		gVisionSensor.OPT.Resolution_mmPerPx		:= gVisionSensor.OPT.FieldOfView_X_mm / gVisionSensor.OPT.ResolutionX;
	ELSE
		gVisionSensor.OPT.PixelSizeBinning_um		:= 0;
		gVisionSensor.OPT.DistanceLens_mm			:= 0;
		gVisionSensor.OPT.CircleOfConfusion_mm		:= 0;
		gVisionSensor.OPT.HyperFocalDistance_mm		:= 0;
		gVisionSensor.OPT.DepthOfFieldNearPos_mm	:= 0;
		gVisionSensor.OPT.DepthOfFieldFarPos_mm		:= 0;
		gVisionSensor.OPT.DepthOfField_mm			:= 0;
		gVisionSensor.OPT.FieldOfView_X_mm			:= 0;
		gVisionSensor.OPT.FieldOfView_Y_mm			:= 0;
		gVisionSensor.OPT.Resolution_mmPerPx		:= 0;
	END_IF

END_PROGRAM
```

#### Vi_main.var - Local variables
```iecst
(*-----------------------------------------------------------------------------------------------------------------------------------------*)
(*Vision function blocks*)
VAR
	ViBaseLoadApplication_01 : ViBaseLoadApplication;
	ViBaseSaveDiagData_01 : ViBaseSaveDiagData;
	FDelete : FileDelete;
END_VAR
(*-----------------------------------------------------------------------------------------------------------------------------------------*)
(*Local variables*)
VAR
	idSensor : UINT := 1;
	TriggerTimeoutSensor : TON; (*Disable web reload when timed out*)
	AcquisitionFailedCntOld : UDINT; (*Old aquisition failed counter*)
	AcquisitionCompletedCntOld : UDINT; (*Old aquisition completed counter*)
	AutoSetupRunning : BOOL; (*Flag for auto setup running*)
END_VAR
(*-----------------------------------------------------------------------------------------------------------------------------------------*)
(*Camera info*)
VAR
	DiagCreateInfo_0 : DiagCreateInfo;
	DiagGetNumInfo_0 : DiagGetNumInfo;
	DiagGetStrInfo_0 : DiagGetStrInfo;
	DiagDisposeInfo_0 : DiagDisposeInfo;
	OpticsReadStep : ARRAY[0..MAX_NUM_CAMS] OF USINT;
	Index : UDINT;
	pChar : REFERENCE TO USINT;
END_VAR
(*Constants*)
VAR CONSTANT
	DISTANCE_FRONTGLASS_LENS_MM : LREAL := 15.0;
	SENSOR_1_3_MP : USINT := 0;
	SENSOR_3_5_MP : USINT := 1;
	SENSOR_5_3_MP : USINT := 2;
	LENS_4_6 : USINT := 0;
	LENS_6_0 : USINT := 1;
	LENS_8_0 : USINT := 2;
	LENS_12_0 : USINT := 3;
	LENS_16_0 : USINT := 4;
	LENS_25_0 : USINT := 5;
	LENS_12_0_MACRO : USINT := 6;
END_VAR
(*-----------------------------------------------------------------------------------------------------------------------------------------*)
(*Image, crosshair data and constants*)
VAR
	i : UINT;
END_VAR
VAR CONSTANT
	HexTab : STRING[16] := '0123456789ABCDEF';
END_VAR
(*-----------------------------------------------------------------------------------------------------------------------------------------*)
(*Error numbers*)
VAR CONSTANT
	ERR_VA_LIST_NUM : UINT := 30000; (*Number of applications exceeds array size*)
END_VAR
VAR
	TON_DelayAfterAutoSetup : TON;
END_VAR
```

### Program Logical/Source/Vision/YourTask (IEC)

#### Variables.var
```iecst
VAR
	startupDelay : TON_10ms; (*Delay startup for mappVision*)
	cmdLoadRecipeAfterBoot : BOOL;
END_VAR
(**)
```

#### Main.st
```iecst
// -----------------------------------------------------------------------------------------------------------
// Use this task to add your own code
// -----------------------------------------------------------------------------------------------------------

// -----------------------------------------------------------------------------------------------------------
// Initialization
// -----------------------------------------------------------------------------------------------------------
PROGRAM _INIT
	// -----------------------------------------------------------------------------------------------------------
	// Delay startup for mappVision
	startupDelay.IN := 1;
	startupDelay.PT := 200;
	REPEAT
		startupDelay();
		UNTIL startupDelay.Q
	END_REPEAT;

	// -----------------------------------------------------------------------------------------------------------
	// Vision sensor configuration
	// -----------------------------------------------------------------------------------------------------------
	gVisionSensor.CFG.VisionFunction		:= enumCoderReader;			// Used to run specific code for this vision function
	gVisionSensor.CFG.PowerlinkNode			:= 1;						// Powerlink node number
	gVisionSensor.CFG.DataStructure			:= ADR(gCodeReader);		// Global structures that holds all data related to this function
	gVisionSensor.CFG.ComponentLink			:= gCameraCodeReading;		// Vision component name defined under mappVision in the configuration view
	gVisionSensor.CFG.ResolutionWidth_X		:= 1280;
	gVisionSensor.CFG.ResolutionHeight_Y	:= 1024;

	cmdLoadRecipeAfterBoot	:= TRUE;

	gParVision.Cam.MaxItemCnt := 1;
	gParVision.Cam.FlashColor := 1;
	gParVision.Cam.FlashSegment := 15;

	gBarCodeReader.Enable	:= TRUE;

END_PROGRAM

// -----------------------------------------------------------------------------------------------------------
// Cyclic part
// -----------------------------------------------------------------------------------------------------------
PROGRAM _CYCLIC

	// -----------------------------------------------------------------------------------------------------------
	// Transfer data when loading a recipe
	IF cmdLoadRecipeAfterBoot THEN
		cmdLoadRecipeAfterBoot := FALSE;

		gVisionSensor.FCT.ApplicationName	:= gParVision.Cam.ApplicationName;
		gVisionSensor.DAT.Exposure			:= gParVision.Cam.Exposure;
		gVisionSensor.DAT.FlashColor		:= gParVision.Cam.FlashColor;
		gVisionSensor.DAT.FlashSegment		:= gParVision.Cam.FlashSegment;
		gVisionSensor.DAT.Focus				:= gParVision.Cam.Focus;
		gVisionSensor.DAT.Gain				:= gParVision.Cam.Gain;
		gVisionSensor.DAT.MaxItemCnt		:= gParVision.Cam.MaxItemCnt;
		gVisionSensor.DAT.Timeout			:= gParVision.Cam.Timeout;
	ELSE
		gParVision.Cam.ApplicationName		:= gVisionSensor.FCT.ApplicationName;
		gParVision.Cam.Exposure				:= gVisionSensor.DAT.Exposure;
		gParVision.Cam.FlashColor			:= gVisionSensor.DAT.FlashColor;
		gParVision.Cam.FlashSegment			:= gVisionSensor.DAT.FlashSegment;
		gParVision.Cam.Focus				:= gVisionSensor.DAT.Focus;
		gParVision.Cam.Gain					:= gVisionSensor.DAT.Gain;
		gParVision.Cam.MaxItemCnt			:= gVisionSensor.DAT.MaxItemCnt;
		gParVision.Cam.Timeout				:= gVisionSensor.DAT.Timeout;
	END_IF

	// -----------------------------------------------------------------------------------------------------------
	// Fire trigger for camera image
	// -----------------------------------------------------------------------------------------------------------
	IF((gBarCodeReader.Trigger OR EDGEPOS(gVisionSensor.DAT.Enable)) AND gVisionSensor.HW.Ready AND NOT gVisionSensor.DAT.ImageProcessingActive) THEN
		// Add default delay and fire trigger
		IF NETTIME_ENABLE THEN
			gVisionSensor.DAT.NettimeDelay := NettimeCurrent_us + NETTIME_DEFAULT_DELAY;
		END_IF
		gVisionSensor.CMD.ImageTrigger	:= TRUE;
		gBarCodeReader.Trigger			:= FALSE;
		gVisionSensor.DAT.Active		:= TRUE;
	END_IF

	gVisionSensor.DAT.Enable 			:= gBarCodeReader.Enable;

	gBarCodeReader.TakeCount 			:= gVisionSensor.DAT.AcquisitionCompletedCnt;
	gBarCodeReader.SerialNumber			:= gCodeReader.BarcodeText[1];
END_PROGRAM
```

- Visualisation Logical/Source/Visu (not shown)

### Program Logical/Source/LibAsMbTCP1_ST/MbApp (IEC)

#### MbApp.st - Implementation code
```iecst
(********************************************************************
 * COPYRIGHT -- Bernecker + Rainer
 ********************************************************************
 * Program: MbApp
 * File: MbApp.st
 * Author: Bernecker + Rainer
 * Created: October 22, 2009
 ********************************************************************
 * Implementation of program MbApp
 ********************************************************************)

PROGRAM _INIT

	(* init values *)
	mb_station 			:= 'IF2.ST40';					(* path to modbus station *)
	register_address	:= 16#2400;						(* register address on modbus station *)
	register_value		:= 2#1010101010101010;			(* register value to write *)
	coil_address		:= 16#0;						(* coils address on modbus station *)
	fub_status			:= 0;							(* status of function blocks *)
	mb_exception		:= 0;							(* modbus exception *)

	instruction			:= mbMFC_WRITE_SINGLE_REGISTER;	(* start instruction *)

END_PROGRAM

PROGRAM _CYCLIC

	(* WORKING STATE MACHINE *)
	CASE (instruction) OF

		mbMFC_WRITE_SINGLE_REGISTER:
			mbWriteSingleRegister_0.enable 			:= 1;
			mbWriteSingleRegister_0.pStation 		:= ADR(mb_station);
			mbWriteSingleRegister_0.startAddress 	:= register_address;
			mbWriteSingleRegister_0.value 			:= register_value;
			mbWriteSingleRegister_0();										(* call function block *)
			IF (mbWriteSingleRegister_0.status <> ERR_FUB_BUSY) THEN
   				fub_status 			:= mbWriteSingleRegister_0.status;
				check_status 		:= TRUE;			(* flag to check status *)
				instruction_ready 	:= TRUE;			(* flag marks instruction "ready" *)
			END_IF

		mbMFC_READ_COILS:
			mbReadCoils_0.enable := 1;
			mbReadCoils_0.pStation := ADR(mb_station);
   			mbReadCoils_0.startAddress := coil_address;
			mbReadCoils_0.nrCoils := 16;
			mbReadCoils_0.pData := ADR(coil_values);
   			mbReadCoils_0.dataSize := SIZEOF(coil_values);
			mbReadCoils_0();												(* call function block *)
   			IF (mbReadCoils_0.status <> ERR_FUB_BUSY) THEN
   				fub_status 			:= mbReadCoils_0.status;
				check_status 		:= TRUE;			(* flag to check status *)
				instruction_ready 	:= TRUE;			(* flag marks instruction "ready" *)
			END_IF

	END_CASE

	(* ERROR HANDLING *)
	IF (check_status) THEN

		CASE fub_status OF

			ERR_OK:
				(* no error *)

			mbERR_EXCEPTION:
				(* modbus station response sent a modbus exception *)
				mbGetLastException_0.enable := 1;
				mbGetLastException_0.pStation := ADR(mb_station);
				mbGetLastException_0();										(* call function block *)
				mb_exception := mbGetLastException_0.mbExcp;

			ELSE
   				(* other error handling *)

		END_CASE

		(* stop checking *)
		check_status := FALSE;
	END_IF

	(* STATE MACHINE CONTROL *)
	IF (instruction_ready AND fub_status = ERR_OK) THEN

		CASE (instruction) OF

			mbMFC_WRITE_SINGLE_REGISTER:
				instruction 		:= mbMFC_READ_COILS;
				instruction_ready 	:= FALSE;

			mbMFC_READ_COILS:
				instruction 		:= mbMFC_WRITE_SINGLE_REGISTER;
				instruction_ready 	:= FALSE;

		END_CASE

	END_IF

END_PROGRAM
```

#### MbApp.var - Local variables
```iecst
(********************************************************************
 * COPYRIGHT -- Bernecker + Rainer
 ********************************************************************
 * Program: MbApp
 * File: MbApp.var
 * Author: Bernecker + Rainer
 * Created: October 22, 2009
 ********************************************************************
 * Local variables of program MbApp
 ********************************************************************)
VAR
	mb_station : STRING[20]; (*path to modbus station*)
	register_address : UINT; (*register address on modbus station*)
	register_value : UINT; (*register value to write*)
	fub_status : UINT; (*status of function blocks*)
	mb_exception : USINT; (*modbus exception*)
	instruction : UDINT; (*start instruction*)
	mbWriteSingleRegister_0 : mbWriteSingleRegister; (*function block structure*)
	check_status : BOOL; (*flag to check status*)
	mbGetLastException_0 : mbGetLastException; (*function block structure*)
	coil_address : UINT; (*coils address on modbus station*)
	mbReadCoils_0 : mbReadCoils; (*function block structure*)
	coil_values : ARRAY[0..15] OF BOOL; (*read data*)
	instruction_ready : BOOL; (*flag marks instruction "ready"*)
END_VAR
```

Listed in the project but not available here: Logical/Libraries/MyTime/Constants.var, Logical/Source/Utility/srvAudit/Types.typ, Logical/Source/Vision/Vi_main/LocalFunctions.fun, Logical/Source/Vision/Vi_main/LocalFunctions.st
